LIN {X 0,Y 199.538,Z 723.393,A -85,B 0,C 180,E1 -21434.273,E2 -21434.273} C_VEL
LIN {X 0,Y 200.491,Z 712.919,A -85,B 0,C 180,E1 -21436.81,E2 -21436.81} C_VEL
LIN {X 0,Y 201.96,Z 700.232,A -85,B 0,C 180,E1 -21439.305,E2 -21439.305} C_VEL
LIN {X 0,Y 203.313,Z 687.711,A -85,B 0,C 180,E1 -21441.281,E2 -21441.281} C_VEL
LIN {X 0,Y 204.53,Z 673.735,A -85,B 0,C 180,E1 -21443.008,E2 -21443.008} C_VEL
LIN {X 0,Y 205.706,Z 659.307,A -85,B 0,C 180,E1 -21444.338,E2 -21444.338} C_VEL
LIN {X 0,Y 207.39,Z 632.291,A -85,B 0,C 180,E1 -21446.071,E2 -21446.071} C_VEL
LIN {X 0,Y 210.434,Z 583.695,A -85,B 0,C 180,E1 -21448.978,E2 -21448.978} C_VEL
LIN {X 0,Y 207.804,Z 555.517,A -85,B 0,C 180,E1 -21450.892,E2 -21450.892} C_VEL
LIN {X 0,Y 206.873,Z 542.727,A -85,B 0,C 180,E1 -21451.758,E2 -21451.758} C_VEL
LIN {X 0,Y 205.476,Z 537.587,A -85,B 0,C 180,E1 -21452.224,E2 -21452.224} C_VEL
LIN {X 0,Y 203.171,Z 526.588,A -85,B 0,C 180,E1 -21456.553,E2 -21456.553} C_VEL
LIN {X 0,Y 200.78,Z 515.899,A -85,B 0,C 180,E1 -21461,E2 -21461} C_VEL
LIN {X 0,Y 199.612,Z 510.746,A -85,B 0,C 180,E1 -21463.319,E2 -21463.319} C_VEL
LIN {X 0,Y 199.581,Z 510.751,A -85,B 0,C 180,E1 -21468.005,E2 -21468.005} C_VEL
LIN {X 0,Y 199.612,Z 510.744,A -85,B 0,C 180,E1 -21470.767,E2 -21470.767} C_VEL
LIN {X 0,Y 199.616,Z 510.742,A -85,B 0,C 180,E1 -21475.714,E2 -21475.714} C_VEL
LIN {X 0,Y 199.703,Z 510.733,A -85,B 0,C 180,E1 -21478.137,E2 -21478.137} C_VEL
LIN {X 0,Y 199.688,Z 510.733,A -85,B 0,C 180,E1 -21482.772,E2 -21482.772} C_VEL
LIN {X 0,Y 199.74,Z 510.729,A -85,B 0,C 180,E1 -21487.229,E2 -21487.229} C_VEL
LIN {X 0,Y 199.798,Z 510.719,A -85,B 0,C 180,E1 -21491.757,E2 -21491.757} C_VEL
LIN {X 0,Y 199.85,Z 510.716,A -85,B 0,C 180,E1 -21495.749,E2 -21495.749} C_VEL
LIN {X 0,Y 200.077,Z 510.684,A -85,B 0,C 180,E1 -21499.884,E2 -21499.884} C_VEL
LIN {X 0,Y 200.134,Z 510.678,A -85,B 0,C 180,E1 -21501.925,E2 -21501.925} C_VEL
LIN {X 0,Y 200.326,Z 510.653,A -85,B 0,C 180,E1 -21507.989,E2 -21507.989} C_VEL
LIN {X 0,Y 200.485,Z 510.633,A -85,B 0,C 180,E1 -21510,E2 -21510} C_VEL
LIN {X 0,Y 200.035,Z 510.692,A -85,B 0,C 180,E1 -21514.029,E2 -21514.029} C_VEL
LIN {X 0,Y 200.134,Z 510.675,A -85,B 0,C 180,E1 -21518.075,E2 -21518.075} C_VEL
LIN {X 0,Y 199.916,Z 510.706,A -85,B 0,C 180,E1 -21522.177,E2 -21522.177} C_VEL
LIN {X 0,Y 199.807,Z 510.716,A -85,B 0,C 180,E1 -21526.343,E2 -21526.343} C_VEL
LIN {X 0,Y 199.825,Z 510.716,A -85,B 0,C 180,E1 -21528.454,E2 -21528.454} C_VEL
LIN {X 0,Y 199.738,Z 510.726,A -85,B 0,C 180,E1 -21533.817,E2 -21533.817} C_VEL
LIN {X 0,Y 199.709,Z 510.731,A -85,B 0,C 180,E1 -21538.384,E2 -21538.384} C_VEL
LIN {X 0,Y 199.659,Z 510.736,A -85,B 0,C 180,E1 -21542.349,E2 -21542.349} C_VEL
LIN {X 0,Y 199.641,Z 510.74,A -85,B 0,C 180,E1 -21546.759,E2 -21546.759} C_VEL
LIN {X 0,Y 199.64,Z 510.743,A -85,B 0,C 180,E1 -21549.321,E2 -21549.321} C_VEL
LIN {X 0,Y 199.583,Z 510.747,A -85,B 0,C 180,E1 -21554.771,E2 -21554.771} C_VEL
LIN {X 0,Y 199.704,Z 510.844,A -85,B 0,C 180,E1 -21560.294,E2 -21560.294} C_VEL
LIN {X 0,Y 203.098,Z 525.538,A -85,B 0,C 180,E1 -21564.592,E2 -21564.592} C_VEL
LIN {X 0,Y 206.826,Z 542.586,A -85,B 0,C 180,E1 -21569.356,E2 -21569.356} C_VEL
LIN {X 0,Y 205.704,Z 551.793,A -85,B 0,C 180,E1 -21571.639,E2 -21571.639} C_VEL
LIN {X 0,Y 207.348,Z 576.297,A -85,B 0,C 180,E1 -21573.193,E2 -21573.193} C_VEL
LIN {X 0,Y 208.243,Z 586.426,A -85,B 0,C 180,E1 -21573.836,E2 -21573.836} C_VEL
LIN {X 0,Y 204.55,Z 659.312,A -85,B 0,C 180,E1 -21578.195,E2 -21578.195} C_VEL
LIN {X 0,Y 203.772,Z 672.943,A -85,B 0,C 180,E1 -21579.255,E2 -21579.255} C_VEL
LIN {X 0,Y 202.728,Z 687.033,A -85,B 0,C 180,E1 -21580.771,E2 -21580.771} C_VEL
LIN {X 0,Y 201.448,Z 700.836,A -85,B 0,C 180,E1 -21582.75,E2 -21582.75} C_VEL
LIN {X 0,Y 200.524,Z 711.943,A -85,B 0,C 180,E1 -21584.76,E2 -21584.76} C_VEL
LIN {X 0,Y 199.491,Z 723.222,A -85,B 0,C 180,E1 -21587.28,E2 -21587.28} C_VEL
LIN {X 0,Y 198.722,Z 732.467,A -85,B 0,C 180,E1 -21589.815,E2 -21589.815} C_VEL
LIN {X 0,Y 198.121,Z 741.455,A -85,B 0,C 180,E1 -21592.869,E2 -21592.869} C_VEL
LIN {X 0,Y 197.748,Z 748.732,A -85,B 0,C 180,E1 -21595.924,E2 -21595.924} C_VEL
LIN {X 0,Y 197.616,Z 754.553,A -85,B 0,C 180,E1 -21598.981,E2 -21598.981} C_VEL
LIN {X 0,Y 197.613,Z 759.139,A -85,B 0,C 180,E1 -21602.038,E2 -21602.038} C_VEL
LIN {X 0,Y 197.951,Z 763.564,A -85,B 0,C 180,E1 -21606.114,E2 -21606.114} C_VEL
LIN {X 0,Y 198.53,Z 765.19,A -85,B 0,C 180,E1 -21608.141,E2 -21608.141} C_VEL
LIN {X 0,Y 200.16,Z 767.195,A -85,B 0,C 180,E1 -21612.162,E2 -21612.162} C_VEL
LIN {X 0,Y 202.917,Z 767.735,A -85,B 0,C 180,E1 -21616.086,E2 -21616.086} C_VEL
LIN {X 0,Y 206.512,Z 766.801,A -85,B 0,C 180,E1 -21619.896,E2 -21619.896} C_VEL
LIN {X 0,Y 211.438,Z 764.341,A -85,B 0,C 180,E1 -21623.508,E2 -21623.508} C_VEL
LIN {X 0,Y 215.761,Z 761.475,A -85,B 0,C 180,E1 -21626.087,E2 -21626.087} C_VEL
LIN {X 0,Y 220.617,Z 757.719,A -85,B 0,C 180,E1 -21628.545,E2 -21628.545} C_VEL
LIN {X 0,Y 227.825,Z 751.158,A -85,B 0,C 180,E1 -21631.629,E2 -21631.629} C_VEL
LIN {X 0,Y 233.763,Z 744.904,A -85,B 0,C 180,E1 -21633.793,E2 -21633.793} C_VEL
LIN {X 0,Y 241.273,Z 736.006,A -85,B 0,C 180,E1 -21636.147,E2 -21636.147} C_VEL
LIN {X 0,Y 248.109,Z 726.715,A -85,B 0,C 180,E1 -21638.032,E2 -21638.032} C_VEL
LIN {X 0,Y 254.857,Z 716.208,A -85,B 0,C 180,E1 -21639.646,E2 -21639.646} C_VEL
LIN {X 0,Y 261.182,Z 704.933,A -85,B 0,C 180,E1 -21640.987,E2 -21640.987} C_VEL
LIN {X 0,Y 263.869,Z 699.471,A -85,B 0,C 180,E1 -21641.52,E2 -21641.52} C_VEL
LIN {X 0,Y 264.318,Z 698.406,A -85,B 0,C 180,E1 -21641.773,E2 -21641.773} C_VEL
LIN {X 0,Y 264.338,Z 697.972,A -85,B 0,C 180,E1 -21642.395,E2 -21642.395} C_VEL
LIN {X 0,Y 263.457,Z 699.205,A -85,B 0,C 180,E1 -21643.374,E2 -21643.374} C_VEL
LIN {X 0,Y 262.431,Z 700.943,A -85,B 0,C 180,E1 -21644.031,E2 -21644.031} C_VEL
LIN {X 0,Y 259.901,Z 705.499,A -85,B 0,C 180,E1 -21645.208,E2 -21645.208} C_VEL
LIN {X 0,Y 257.019,Z 710.646,A -85,B 0,C 180,E1 -21646.213,E2 -21646.213} C_VEL
LIN {X 0,Y 254.784,Z 714.396,A -85,B 0,C 180,E1 -21646.735,E2 -21646.735} C_VEL
LIN {X 0,Y 247.204,Z 725.947,A -85,B 0,C 180,E1 -21648.238,E2 -21648.238} C_VEL
LIN {X 0,Y 238.723,Z 737.138,A -85,B 0,C 180,E1 -21650.184,E2 -21650.184} C_VEL
LIN {X 0,Y 231.018,Z 746.108,A -85,B 0,C 180,E1 -21652.276,E2 -21652.276} C_VEL
LIN {X 0,Y 223.904,Z 753.524,A -85,B 0,C 180,E1 -21654.501,E2 -21654.501} C_VEL
LIN {X 0,Y 217.848,Z 759.259,A -85,B 0,C 180,E1 -21656.74,E2 -21656.74} C_VEL
LIN {X 0,Y 210.681,Z 765.375,A -85,B 0,C 180,E1 -21659.975,E2 -21659.975} C_VEL
LIN {X 0,Y 204.411,Z 769.92,A -85,B 0,C 180,E1 -21663.451,E2 -21663.451} C_VEL
LIN {X 0,Y 199.387,Z 773.014,A -85,B 0,C 180,E1 -21667.187,E2 -21667.187} C_VEL
LIN {X 0,Y 195.455,Z 774.755,A -85,B 0,C 180,E1 -21671.118,E2 -21671.118} C_VEL
LIN {X 0,Y 192.647,Z 775.104,A -85,B 0,C 180,E1 -21675.205,E2 -21675.205} C_VEL
LIN {X 0,Y 191.118,Z 774.041,A -85,B 0,C 180,E1 -21679.405,E2 -21679.405} C_VEL
LIN {X 0,Y 190.659,Z 771.533,A -85,B 0,C 180,E1 -21683.651,E2 -21683.651} C_VEL
LIN {X 0,Y 190.784,Z 768.594,A -85,B 0,C 180,E1 -21686.833,E2 -21686.833} C_VEL
LIN {X 0,Y 191.06,Z 766.027,A -85,B 0,C 180,E1 -21689.078,E2 -21689.078} C_VEL
LIN {X 0,Y 190.744,Z 769.407,A -85,B 0,C 180,E1 -21692.112,E2 -21692.112} C_VEL
LIN {X 0,Y 190.574,Z 772.03,A -85,B 0,C 180,E1 -21695.311,E2 -21695.311} C_VEL
LIN {X 0,Y 190.623,Z 773.843,A -85,B 0,C 180,E1 -21698.481,E2 -21698.481} C_VEL
LIN {X 0,Y 191.584,Z 775.164,A -85,B 0,C 180,E1 -21702.715,E2 -21702.715} C_VEL
LIN {X 0,Y 193.65,Z 775.273,A -85,B 0,C 180,E1 -21706.878,E2 -21706.878} C_VEL
LIN {X 0,Y 196.855,Z 774.188,A -85,B 0,C 180,E1 -21710.917,E2 -21710.917} C_VEL
LIN {X 0,Y 201.1,Z 771.909,A -85,B 0,C 180,E1 -21714.795,E2 -21714.795} C_VEL
LIN {X 0,Y 206.36,Z 768.461,A -85,B 0,C 180,E1 -21718.477,E2 -21718.477} C_VEL
LIN {X 0,Y 212.807,Z 763.716,A -85,B 0,C 180,E1 -21721.898,E2 -21721.898} C_VEL
LIN {X 0,Y 220.248,Z 757.558,A -85,B 0,C 180,E1 -21725.056,E2 -21725.056} C_VEL
LIN {X 0,Y 227.423,Z 751.033,A -85,B 0,C 180,E1 -21727.614,E2 -21727.614} C_VEL
LIN {X 0,Y 236.499,Z 741.882,A -85,B 0,C 180,E1 -21730.267,E2 -21730.267} C_VEL
LIN {X 0,Y 243.795,Z 733.654,A -85,B 0,C 180,E1 -21732.086,E2 -21732.086} C_VEL
LIN {X 0,Y 252.794,Z 722.394,A -85,B 0,C 180,E1 -21734.03,E2 -21734.03} C_VEL
LIN {X 0,Y 261.497,Z 709.921,A -85,B 0,C 180,E1 -21735.627,E2 -21735.627} C_VEL
LIN {X 0,Y 267.73,Z 699.805,A -85,B 0,C 180,E1 -21736.599,E2 -21736.599} C_VEL
LIN {X 0,Y 269.637,Z 696.414,A -85,B 0,C 180,E1 -21736.871,E2 -21736.871} C_VEL
LIN {X 0,Y 268.965,Z 697.521,A -85,B 0,C 180,E1 -21737.205,E2 -21737.205} C_VEL
LIN {X 0,Y 261.172,Z 710.023,A -85,B 0,C 180,E1 -21738.498,E2 -21738.498} C_VEL
LIN {X 0,Y 252.468,Z 722.025,A -85,B 0,C 180,E1 -21740.189,E2 -21740.189} C_VEL
LIN {X 0,Y 244.82,Z 731.27,A -85,B 0,C 180,E1 -21741.888,E2 -21741.888} C_VEL
LIN {X 0,Y 236.371,Z 740.349,A -85,B 0,C 180,E1 -21744.04,E2 -21744.04} C_VEL
LIN {X 0,Y 227.276,Z 748.967,A -85,B 0,C 180,E1 -21746.829,E2 -21746.829} C_VEL
LIN {X 0,Y 220.355,Z 754.627,A -85,B 0,C 180,E1 -21749.316,E2 -21749.316} C_VEL
LIN {X 0,Y 214.842,Z 758.693,A -85,B 0,C 180,E1 -21751.684,E2 -21751.684} C_VEL
LIN {X 0,Y 209.813,Z 761.867,A -85,B 0,C 180,E1 -21754.186,E2 -21754.186} C_VEL
LIN {X 0,Y 204.001,Z 764.903,A -85,B 0,C 180,E1 -21757.731,E2 -21757.731} C_VEL
LIN {X 0,Y 199.095,Z 766.562,A -85,B 0,C 180,E1 -21761.476,E2 -21761.476} C_VEL
LIN {X 0,Y 195.476,Z 766.806,A -85,B 0,C 180,E1 -21765.423,E2 -21765.423} C_VEL
LIN {X 0,Y 192.791,Z 765.642,A -85,B 0,C 180,E1 -21769.498,E2 -21769.498} C_VEL
LIN {X 0,Y 191.187,Z 763.064,A -85,B 0,C 180,E1 -21773.669,E2 -21773.669} C_VEL
LIN {X 0,Y 190.614,Z 758.971,A -85,B 0,C 180,E1 -21777.887,E2 -21777.887} C_VEL
LIN {X 0,Y 190.501,Z 754.761,A -85,B 0,C 180,E1 -21781.057,E2 -21781.057} C_VEL
LIN {X 0,Y 190.533,Z 749.385,A -85,B 0,C 180,E1 -21784.231,E2 -21784.231} C_VEL
LIN {X 0,Y 190.87,Z 742.738,A -85,B 0,C 180,E1 -21787.404,E2 -21787.404} C_VEL
LIN {X 0,Y 191.407,Z 734.574,A -85,B 0,C 180,E1 -21790.579,E2 -21790.579} C_VEL
LIN {X 0,Y 192.322,Z 724.548,A -85,B 0,C 180,E1 -21793.741,E2 -21793.741} C_VEL
LIN {X 0,Y 193.237,Z 714.276,A -85,B 0,C 180,E1 -21796.372,E2 -21796.372} C_VEL
LIN {X 0,Y 194.667,Z 701.848,A -85,B 0,C 180,E1 -21798.961,E2 -21798.961} C_VEL
LIN {X 0,Y 196.017,Z 689.687,A -85,B 0,C 180,E1 -21801.011,E2 -21801.011} C_VEL
LIN {X 0,Y 197.215,Z 676.294,A -85,B 0,C 180,E1 -21802.801,E2 -21802.801} C_VEL
LIN {X 0,Y 198.466,Z 661.566,A -85,B 0,C 180,E1 -21804.309,E2 -21804.309} C_VEL
LIN {X 0,Y 199.852,Z 640.548,A -85,B 0,C 180,E1 -21805.797,E2 -21805.797} C_VEL
LIN {X 0,Y 203.424,Z 584.022,A -85,B 0,C 180,E1 -21809.337,E2 -21809.337} C_VEL
LIN {X 0,Y 200.675,Z 552.776,A -85,B 0,C 180,E1 -21811.545,E2 -21811.545} C_VEL
LIN {X 0,Y 200.037,Z 544.275,A -85,B 0,C 180,E1 -21812.141,E2 -21812.141} C_VEL
LIN {X 0,Y 198.245,Z 537.538,A -85,B 0,C 180,E1 -21812.733,E2 -21812.733} C_VEL
LIN {X 0,Y 195.977,Z 526.924,A -85,B 0,C 180,E1 -21817.07,E2 -21817.07} C_VEL
LIN {X 0,Y 193.455,Z 515.636,A -85,B 0,C 180,E1 -21821.947,E2 -21821.947} C_VEL
LIN {X 0,Y 192.558,Z 511.625,A -85,B 0,C 180,E1 -21823.748,E2 -21823.748} C_VEL
LIN {X 0,Y 192.515,Z 511.63,A -85,B 0,C 180,E1 -21828.92,E2 -21828.92} C_VEL
LIN {X 0,Y 192.588,Z 511.621,A -85,B 0,C 180,E1 -21833.402,E2 -21833.402} C_VEL
LIN {X 0,Y 192.612,Z 511.614,A -85,B 0,C 180,E1 -21837.058,E2 -21837.058} C_VEL
LIN {X 0,Y 192.666,Z 511.61,A -85,B 0,C 180,E1 -21841.692,E2 -21841.692} C_VEL
LIN {X 0,Y 192.707,Z 511.603,A -85,B 0,C 180,E1 -21846.349,E2 -21846.349} C_VEL
LIN {X 0,Y 192.733,Z 511.6,A -85,B 0,C 180,E1 -21851.457,E2 -21851.457} C_VEL
LIN {X 0,Y 192.774,Z 511.596,A -85,B 0,C 180,E1 -21855.214,E2 -21855.214} C_VEL
LIN {X 0,Y 193.022,Z 511.565,A -85,B 0,C 180,E1 -21859.51,E2 -21859.51} C_VEL
LIN {X 0,Y 193.007,Z 511.568,A -85,B 0,C 180,E1 -21863.728,E2 -21863.728} C_VEL
LIN {X 0,Y 193.268,Z 511.533,A -85,B 0,C 180,E1 -21867.916,E2 -21867.916} C_VEL
LIN {X 0,Y 193.448,Z 511.509,A -85,B 0,C 180,E1 -21870,E2 -21870} C_VEL
LIN {X 0,Y 192.982,Z 511.57,A -85,B 0,C 180,E1 -21874.177,E2 -21874.177} C_VEL
LIN {X 0,Y 193.081,Z 511.553,A -85,B 0,C 180,E1 -21878.372,E2 -21878.372} C_VEL
LIN {X 0,Y 192.855,Z 511.586,A -85,B 0,C 180,E1 -21882.63,E2 -21882.63} C_VEL
LIN {X 0,Y 192.782,Z 511.593,A -85,B 0,C 180,E1 -21888.586,E2 -21888.586} C_VEL
LIN {X 0,Y 192.665,Z 511.606,A -85,B 0,C 180,E1 -21894.225,E2 -21894.225} C_VEL
LIN {X 0,Y 192.645,Z 511.612,A -85,B 0,C 180,E1 -21898.889,E2 -21898.889} C_VEL
LIN {X 0,Y 192.599,Z 511.616,A -85,B 0,C 180,E1 -21903.186,E2 -21903.186} C_VEL
LIN {X 0,Y 192.61,Z 511.616,A -85,B 0,C 180,E1 -21906.608,E2 -21906.608} C_VEL
LIN {X 0,Y 192.525,Z 511.627,A -85,B 0,C 180,E1 -21911.077,E2 -21911.077} C_VEL
LIN {X 0,Y 192.494,Z 511.631,A -85,B 0,C 180,E1 -21916.077,E2 -21916.077} C_VEL
LIN {X 0,Y 192.647,Z 511.756,A -85,B 0,C 180,E1 -21919.857,E2 -21919.857} C_VEL
LIN {X 0,Y 196.065,Z 526.547,A -85,B 0,C 180,E1 -21924.291,E2 -21924.291} C_VEL
LIN {X 0,Y 199.703,Z 543.053,A -85,B 0,C 180,E1 -21929.027,E2 -21929.027} C_VEL
LIN {X 0,Y 198.736,Z 551.747,A -85,B 0,C 180,E1 -21931.279,E2 -21931.279} C_VEL
LIN {X 0,Y 200.206,Z 575.588,A -85,B 0,C 180,E1 -21932.848,E2 -21932.848} C_VEL
LIN {X 0,Y 201.175,Z 587.238,A -85,B 0,C 180,E1 -21933.62,E2 -21933.62} C_VEL
LIN {X 0,Y 197.436,Z 659.441,A -85,B 0,C 180,E1 -21938.166,E2 -21938.166} C_VEL
LIN {X 0,Y 196.622,Z 673.729,A -85,B 0,C 180,E1 -21939.331,E2 -21939.331} C_VEL
LIN {X 0,Y 195.6,Z 687.334,A -85,B 0,C 180,E1 -21940.861,E2 -21940.861} C_VEL
LIN {X 0,Y 194.328,Z 701.111,A -85,B 0,C 180,E1 -21942.912,E2 -21942.912} C_VEL
LIN {X 0,Y 193.391,Z 712.142,A -85,B 0,C 180,E1 -21944.994,E2 -21944.994} C_VEL
LIN {X 0,Y 192.369,Z 723.29,A -85,B 0,C 180,E1 -21947.606,E2 -21947.606} C_VEL
LIN {X 0,Y 191.583,Z 733.292,A -85,B 0,C 180,E1 -21950.498,E2 -21950.498} C_VEL
LIN {X 0,Y 191.032,Z 742.187,A -85,B 0,C 180,E1 -21953.663,E2 -21953.663} C_VEL
LIN {X 0,Y 190.726,Z 749.346,A -85,B 0,C 180,E1 -21956.832,E2 -21956.832} C_VEL
LIN {X 0,Y 190.588,Z 755.01,A -85,B 0,C 180,E1 -21960,E2 -21960} C_VEL
LIN {X 0,Y 190.61,Z 759.489,A -85,B 0,C 180,E1 -21963.171,E2 -21963.171} C_VEL
LIN {X 0,Y 190.924,Z 762.954,A -85,B 0,C 180,E1 -21966.34,E2 -21966.34} C_VEL
LIN {X 0,Y 192.242,Z 766.101,A -85,B 0,C 180,E1 -21970.532,E2 -21970.532} C_VEL
LIN {X 0,Y 194.54,Z 767.777,A -85,B 0,C 180,E1 -21974.648,E2 -21974.648} C_VEL
LIN {X 0,Y 197.887,Z 767.941,A -85,B 0,C 180,E1 -21978.641,E2 -21978.641} C_VEL
LIN {X 0,Y 199.901,Z 767.499,A -85,B 0,C 180,E1 -21980.584,E2 -21980.584} C_VEL
LIN {X 0,Y 205.058,Z 765.507,A -85,B 0,C 180,E1 -21984.285,E2 -21984.285} C_VEL
LIN {X 0,Y 207.958,Z 763.962,A -85,B 0,C 180,E1 -21986.062,E2 -21986.062} C_VEL
LIN {X 0,Y 214.603,Z 759.634,A -85,B 0,C 180,E1 -21989.422,E2 -21989.422} C_VEL
LIN {X 0,Y 220.177,Z 755.324,A -85,B 0,C 180,E1 -21991.781,E2 -21991.781} C_VEL
LIN {X 0,Y 227.232,Z 749.022,A -85,B 0,C 180,E1 -21994.364,E2 -21994.364} C_VEL
LIN {X 0,Y 234.899,Z 741.08,A -85,B 0,C 180,E1 -21996.754,E2 -21996.754} C_VEL
LIN {X 0,Y 241.856,Z 732.883,A -85,B 0,C 180,E1 -21998.665,E2 -21998.665} C_VEL
LIN {X 0,Y 249.347,Z 722.876,A -85,B 0,C 180,E1 -22000.411,E2 -22000.411} C_VEL
LIN {X 0,Y 256.515,Z 711.735,A -85,B 0,C 180,E1 -22001.9,E2 -22001.9} C_VEL
LIN {X 0,Y 262.946,Z 700.024,A -85,B 0,C 180,E1 -22003.08,E2 -22003.08} C_VEL
LIN {X 0,Y 268.228,Z 688.618,A -85,B 0,C 180,E1 -22003.975,E2 -22003.975} C_VEL
LIN {X 0,Y 269.024,Z 686.717,A -85,B 0,C 180,E1 -22004.102,E2 -22004.102} C_VEL
LIN {X 0,Y 269.42,Z 685.699,A -85,B 0,C 180,E1 -22004.443,E2 -22004.443} C_VEL
LIN {X 0,Y 263.476,Z 698.717,A -85,B 0,C 180,E1 -22005.289,E2 -22005.289} C_VEL
LIN {X 0,Y 257.055,Z 710.637,A -85,B 0,C 180,E1 -22006.342,E2 -22006.342} C_VEL
LIN {X 0,Y 254.784,Z 714.396,A -85,B 0,C 180,E1 -22006.735,E2 -22006.735} C_VEL
LIN {X 0,Y 251.69,Z 719.15,A -85,B 0,C 180,E1 -22007.147,E2 -22007.147} C_VEL
LIN {X 0,Y 245.838,Z 727.009,A -85,B 0,C 180,E1 -22007.524,E2 -22007.524} C_VEL
LIN {X 0,Y 239.679,Z 734.365,A -85,B 0,C 180,E1 -22008.005,E2 -22008.005} C_VEL
LIN {X 0,Y 236.142,Z 738.329,A -85,B 0,C 180,E1 -22008.587,E2 -22008.587} C_VEL
LIN {X 0,Y 227.616,Z 747.405,A -85,B 0,C 180,E1 -22010.73,E2 -22010.73} C_VEL
LIN {X 0,Y 220.62,Z 754.006,A -85,B 0,C 180,E1 -22012.752,E2 -22012.752} C_VEL
LIN {X 0,Y 214.164,Z 759.568,A -85,B 0,C 180,E1 -22014.951,E2 -22014.951} C_VEL
LIN {X 0,Y 208.291,Z 764.134,A -85,B 0,C 180,E1 -22017.326,E2 -22017.326} C_VEL
LIN {X 0,Y 201.283,Z 768.901,A -85,B 0,C 180,E1 -22020.737,E2 -22020.737} C_VEL
LIN {X 0,Y 195.34,Z 772.234,A -85,B 0,C 180,E1 -22024.422,E2 -22024.422} C_VEL
LIN {X 0,Y 190.648,Z 774.189,A -85,B 0,C 180,E1 -22028.368,E2 -22028.368} C_VEL
LIN {X 0,Y 187.113,Z 774.819,A -85,B 0,C 180,E1 -22032.514,E2 -22032.514} C_VEL
LIN {X 0,Y 184.858,Z 774.114,A -85,B 0,C 180,E1 -22036.814,E2 -22036.814} C_VEL
LIN {X 0,Y 183.783,Z 771.993,A -85,B 0,C 180,E1 -22041.201,E2 -22041.201} C_VEL
LIN {X 0,Y 183.786,Z 768.349,A -85,B 0,C 180,E1 -22045.614,E2 -22045.614} C_VEL
LIN {X 0,Y 184.114,Z 764.515,A -85,B 0,C 180,E1 -22049.043,E2 -22049.043} C_VEL
LIN {X 0,Y 183.694,Z 769.129,A -85,B 0,C 180,E1 -22053.29,E2 -22053.29} C_VEL
LIN {X 0,Y 183.514,Z 771.696,A -85,B 0,C 180,E1 -22056.597,E2 -22056.597} C_VEL
LIN {X 0,Y 184.062,Z 773.925,A -85,B 0,C 180,E1 -22061.006,E2 -22061.006} C_VEL
LIN {X 0,Y 185.559,Z 774.936,A -85,B 0,C 180,E1 -22065.375,E2 -22065.375} C_VEL
LIN {X 0,Y 188.401,Z 774.77,A -85,B 0,C 180,E1 -22069.617,E2 -22069.617} C_VEL
LIN {X 0,Y 192.278,Z 773.441,A -85,B 0,C 180,E1 -22073.708,E2 -22073.708} C_VEL
LIN {X 0,Y 197.392,Z 770.954,A -85,B 0,C 180,E1 -22077.572,E2 -22077.572} C_VEL
LIN {X 0,Y 203.443,Z 767.313,A -85,B 0,C 180,E1 -22081.21,E2 -22081.21} C_VEL
LIN {X 0,Y 210.669,Z 762.373,A -85,B 0,C 180,E1 -22084.55,E2 -22084.55} C_VEL
LIN {X 0,Y 218.805,Z 756.107,A -85,B 0,C 180,E1 -22087.61,E2 -22087.61} C_VEL
LIN {X 0,Y 227.831,Z 748.331,A -85,B 0,C 180,E1 -22090.376,E2 -22090.376} C_VEL
LIN {X 0,Y 237.647,Z 738.718,A -85,B 0,C 180,E1 -22092.859,E2 -22092.859} C_VEL
LIN {X 0,Y 245.49,Z 730.127,A -85,B 0,C 180,E1 -22094.54,E2 -22094.54} C_VEL
LIN {X 0,Y 253.719,Z 720.134,A -85,B 0,C 180,E1 -22096.071,E2 -22096.071} C_VEL
LIN {X 0,Y 259.381,Z 712.449,A -85,B 0,C 180,E1 -22097.019,E2 -22097.019} C_VEL
LIN {X 0,Y 254.554,Z 718.823,A -85,B 0,C 180,E1 -22097.917,E2 -22097.917} C_VEL
LIN {X 0,Y 246.269,Z 728.621,A -85,B 0,C 180,E1 -22099.516,E2 -22099.516} C_VEL
LIN {X 0,Y 237.221,Z 738.14,A -85,B 0,C 180,E1 -22101.526,E2 -22101.526} C_VEL
LIN {X 0,Y 228.736,Z 745.987,A -85,B 0,C 180,E1 -22103.739,E2 -22103.739} C_VEL
LIN {X 0,Y 220.253,Z 752.791,A -85,B 0,C 180,E1 -22106.333,E2 -22106.333} C_VEL
LIN {X 0,Y 212.546,Z 758.198,A -85,B 0,C 180,E1 -22109.168,E2 -22109.168} C_VEL
LIN {X 0,Y 206.989,Z 761.576,A -85,B 0,C 180,E1 -22111.618,E2 -22111.618} C_VEL
LIN {X 0,Y 200.447,Z 764.78,A -85,B 0,C 180,E1 -22115.119,E2 -22115.119} C_VEL
LIN {X 0,Y 194.867,Z 766.667,A -85,B 0,C 180,E1 -22118.859,E2 -22118.859} C_VEL
LIN {X 0,Y 190.322,Z 767.202,A -85,B 0,C 180,E1 -22122.817,E2 -22122.817} C_VEL
LIN {X 0,Y 187.097,Z 766.38,A -85,B 0,C 180,E1 -22126.975,E2 -22126.975} C_VEL
LIN {X 0,Y 184.841,Z 764.169,A -85,B 0,C 180,E1 -22131.252,E2 -22131.252} C_VEL
LIN {X 0,Y 183.796,Z 760.491,A -85,B 0,C 180,E1 -22135.614,E2 -22135.614} C_VEL
LIN {X 0,Y 183.525,Z 756.679,A -85,B 0,C 180,E1 -22138.903,E2 -22138.903} C_VEL
LIN {X 0,Y 183.469,Z 751.805,A -85,B 0,C 180,E1 -22142.195,E2 -22142.195} C_VEL
LIN {X 0,Y 183.677,Z 745.06,A -85,B 0,C 180,E1 -22145.822,E2 -22145.822} C_VEL
LIN {X 0,Y 184.183,Z 736.79,A -85,B 0,C 180,E1 -22149.333,E2 -22149.333} C_VEL
LIN {X 0,Y 184.937,Z 727.264,A -85,B 0,C 180,E1 -22152.622,E2 -22152.622} C_VEL
LIN {X 0,Y 185.945,Z 716.545,A -85,B 0,C 180,E1 -22155.622,E2 -22155.622} C_VEL
LIN {X 0,Y 187.18,Z 704.739,A -85,B 0,C 180,E1 -22158.328,E2 -22158.328} C_VEL
LIN {X 0,Y 188.61,Z 692.172,A -85,B 0,C 180,E1 -22160.624,E2 -22160.624} C_VEL
LIN {X 0,Y 189.911,Z 678.748,A -85,B 0,C 180,E1 -22162.576,E2 -22162.576} C_VEL
LIN {X 0,Y 191.114,Z 664.628,A -85,B 0,C 180,E1 -22164.149,E2 -22164.149} C_VEL
LIN {X 0,Y 192.222,Z 649.678,A -85,B 0,C 180,E1 -22165.37,E2 -22165.37} C_VEL
LIN {X 0,Y 196.444,Z 584.623,A -85,B 0,C 180,E1 -22169.68,E2 -22169.68} C_VEL
LIN {X 0,Y 193.939,Z 555.999,A -85,B 0,C 180,E1 -22171.772,E2 -22171.772} C_VEL
LIN {X 0,Y 193.238,Z 546.026,A -85,B 0,C 180,E1 -22172.5,E2 -22172.5} C_VEL
LIN {X 0,Y 190.956,Z 537.385,A -85,B 0,C 180,E1 -22173.306,E2 -22173.306} C_VEL
LIN {X 0,Y 188.38,Z 525.374,A -85,B 0,C 180,E1 -22178.421,E2 -22178.421} C_VEL
LIN {X 0,Y 186.035,Z 514.853,A -85,B 0,C 180,E1 -22183.167,E2 -22183.167} C_VEL
LIN {X 0,Y 185.496,Z 512.504,A -85,B 0,C 180,E1 -22184.357,E2 -22184.357} C_VEL
LIN {X 0,Y 185.47,Z 512.508,A -85,B 0,C 180,E1 -22189.895,E2 -22189.895} C_VEL
LIN {X 0,Y 185.507,Z 512.501,A -85,B 0,C 180,E1 -22192.711,E2 -22192.711} C_VEL
LIN {X 0,Y 185.548,Z 512.496,A -85,B 0,C 180,E1 -22197.975,E2 -22197.975} C_VEL
LIN {X 0,Y 185.583,Z 512.491,A -85,B 0,C 180,E1 -22200.576,E2 -22200.576} C_VEL
LIN {X 0,Y 185.589,Z 512.489,A -85,B 0,C 180,E1 -22205.382,E2 -22205.382} C_VEL
LIN {X 0,Y 185.676,Z 512.48,A -85,B 0,C 180,E1 -22211.133,E2 -22211.133} C_VEL
LIN {X 0,Y 185.726,Z 512.472,A -85,B 0,C 180,E1 -22214.64,E2 -22214.64} C_VEL
LIN {X 0,Y 185.944,Z 512.448,A -85,B 0,C 180,E1 -22219.328,E2 -22219.328} C_VEL
LIN {X 0,Y 185.971,Z 512.444,A -85,B 0,C 180,E1 -22223.49,E2 -22223.49} C_VEL
LIN {X 0,Y 186.212,Z 512.412,A -85,B 0,C 180,E1 -22227.837,E2 -22227.837} C_VEL
LIN {X 0,Y 186.411,Z 512.385,A -85,B 0,C 180,E1 -22230,E2 -22230} C_VEL
LIN {X 0,Y 185.93,Z 512.448,A -85,B 0,C 180,E1 -22234.335,E2 -22234.335} C_VEL
LIN {X 0,Y 186.031,Z 512.431,A -85,B 0,C 180,E1 -22238.691,E2 -22238.691} C_VEL
LIN {X 0,Y 185.767,Z 512.47,A -85,B 0,C 180,E1 -22243.12,E2 -22243.12} C_VEL
LIN {X 0,Y 185.718,Z 512.474,A -85,B 0,C 180,E1 -22247.622,E2 -22247.622} C_VEL
LIN {X 0,Y 185.601,Z 512.489,A -85,B 0,C 180,E1 -22252.251,E2 -22252.251} C_VEL
LIN {X 0,Y 185.561,Z 512.493,A -85,B 0,C 180,E1 -22257.032,E2 -22257.032} C_VEL
LIN {X 0,Y 185.578,Z 512.494,A -85,B 0,C 180,E1 -22259.493,E2 -22259.493} C_VEL
LIN {X 0,Y 185.519,Z 512.496,A -85,B 0,C 180,E1 -22264.628,E2 -22264.628} C_VEL
LIN {X 0,Y 185.545,Z 512.499,A -85,B 0,C 180,E1 -22267.304,E2 -22267.304} C_VEL
LIN {X 0,Y 185.487,Z 512.503,A -85,B 0,C 180,E1 -22270.73,E2 -22270.73} C_VEL
LIN {X 0,Y 185.483,Z 512.503,A -85,B 0,C 180,E1 -22273.953,E2 -22273.953} C_VEL
LIN {X 0,Y 185.567,Z 512.52,A -85,B 0,C 180,E1 -22279.369,E2 -22279.369} C_VEL
LIN {X 0,Y 189.206,Z 528.348,A -85,B 0,C 180,E1 -22284.24,E2 -22284.24} C_VEL
LIN {X 0,Y 192.59,Z 543.697,A -85,B 0,C 180,E1 -22288.747,E2 -22288.747} C_VEL
LIN {X 0,Y 192.152,Z 549.113,A -85,B 0,C 180,E1 -22290.201,E2 -22290.201} C_VEL
LIN {X 0,Y 191.735,Z 551.898,A -85,B 0,C 180,E1 -22290.936,E2 -22290.936} C_VEL
LIN {X 0,Y 193.19,Z 576.268,A -85,B 0,C 180,E1 -22292.624,E2 -22292.624} C_VEL
LIN {X 0,Y 194.111,Z 587.271,A -85,B 0,C 180,E1 -22293.381,E2 -22293.381} C_VEL
LIN {X 0,Y 190.376,Z 658.875,A -85,B 0,C 180,E1 -22298.087,E2 -22298.087} C_VEL
LIN {X 0,Y 189.591,Z 672.752,A -85,B 0,C 180,E1 -22299.239,E2 -22299.239} C_VEL
LIN {X 0,Y 188.479,Z 687.413,A -85,B 0,C 180,E1 -22300.957,E2 -22300.957} C_VEL
LIN {X 0,Y 187.235,Z 701.052,A -85,B 0,C 180,E1 -22303.088,E2 -22303.088} C_VEL
LIN {X 0,Y 186.325,Z 712.08,A -85,B 0,C 180,E1 -22305.25,E2 -22305.25} C_VEL
LIN {X 0,Y 185.276,Z 723.249,A -85,B 0,C 180,E1 -22307.958,E2 -22307.958} C_VEL
LIN {X 0,Y 184.562,Z 732.49,A -85,B 0,C 180,E1 -22310.687,E2 -22310.687} C_VEL
LIN {X 0,Y 184.029,Z 741.513,A -85,B 0,C 180,E1 -22313.977,E2 -22313.977} C_VEL
LIN {X 0,Y 183.731,Z 748.746,A -85,B 0,C 180,E1 -22317.259,E2 -22317.259} C_VEL
LIN {X 0,Y 183.604,Z 753.663,A -85,B 0,C 180,E1 -22320,E2 -22320} C_VEL
LIN {X 0,Y 183.613,Z 758.478,A -85,B 0,C 180,E1 -22323.291,E2 -22323.291} C_VEL
LIN {X 0,Y 183.92,Z 762.172,A -85,B 0,C 180,E1 -22326.583,E2 -22326.583} C_VEL
LIN {X 0,Y 185.292,Z 765.747,A -85,B 0,C 180,E1 -22330.932,E2 -22330.932} C_VEL
LIN {X 0,Y 187.676,Z 767.747,A -85,B 0,C 180,E1 -22335.197,E2 -22335.197} C_VEL
LIN {X 0,Y 191.184,Z 768.346,A -85,B 0,C 180,E1 -22339.32,E2 -22339.32} C_VEL
LIN {X 0,Y 193.322,Z 768.125,A -85,B 0,C 180,E1 -22341.318,E2 -22341.318} C_VEL
LIN {X 0,Y 198.696,Z 766.568,A -85,B 0,C 180,E1 -22345.116,E2 -22345.116} C_VEL
LIN {X 0,Y 205.081,Z 763.546,A -85,B 0,C 180,E1 -22348.671,E2 -22348.671} C_VEL
LIN {X 0,Y 210.53,Z 760.275,A -85,B 0,C 180,E1 -22351.16,E2 -22351.16} C_VEL
LIN {X 0,Y 218.506,Z 754.528,A -85,B 0,C 180,E1 -22354.254,E2 -22354.254} C_VEL
LIN {X 0,Y 227.362,Z 746.874,A -85,B 0,C 180,E1 -22357.068,E2 -22357.068} C_VEL
LIN {X 0,Y 235.64,Z 738.504,A -85,B 0,C 180,E1 -22359.33,E2 -22359.33} C_VEL
LIN {X 0,Y 242.851,Z 730.146,A -85,B 0,C 180,E1 -22361.025,E2 -22361.025} C_VEL
LIN {X 0,Y 250.809,Z 719.667,A -85,B 0,C 180,E1 -22362.632,E2 -22362.632} C_VEL
LIN {X 0,Y 258.517,Z 707.672,A -85,B 0,C 180,E1 -22364.023,E2 -22364.023} C_VEL
LIN {X 0,Y 258.314,Z 708,A -85,B 0,C 180,E1 -22364.423,E2 -22364.423} C_VEL
LIN {X 0,Y 250.363,Z 720.249,A -85,B 0,C 180,E1 -22365.711,E2 -22365.711} C_VEL
LIN {X 0,Y 244.16,Z 728.642,A -85,B 0,C 180,E1 -22366.872,E2 -22366.872} C_VEL
LIN {X 0,Y 236.142,Z 738.329,A -85,B 0,C 180,E1 -22368.587,E2 -22368.587} C_VEL
LIN {X 0,Y 232.44,Z 742.224,A -85,B 0,C 180,E1 -22369.236,E2 -22369.236} C_VEL
LIN {X 0,Y 225.43,Z 748.557,A -85,B 0,C 180,E1 -22370.041,E2 -22370.041} C_VEL
LIN {X 0,Y 218.338,Z 754.194,A -85,B 0,C 180,E1 -22370.994,E2 -22370.994} C_VEL
LIN {X 0,Y 214.569,Z 757.075,A -85,B 0,C 180,E1 -22371.875,E2 -22371.875} C_VEL
LIN {X 0,Y 206.485,Z 763.013,A -85,B 0,C 180,E1 -22374.646,E2 -22374.646} C_VEL
LIN {X 0,Y 198.726,Z 767.907,A -85,B 0,C 180,E1 -22377.962,E2 -22377.962} C_VEL
LIN {X 0,Y 191.905,Z 771.434,A -85,B 0,C 180,E1 -22381.57,E2 -22381.57} C_VEL
LIN {X 0,Y 186.401,Z 773.631,A -85,B 0,C 180,E1 -22385.497,E2 -22385.497} C_VEL
LIN {X 0,Y 182.041,Z 774.495,A -85,B 0,C 180,E1 -22389.668,E2 -22389.668} C_VEL
LIN {X 0,Y 178.932,Z 774.039,A -85,B 0,C 180,E1 -22394.041,E2 -22394.041} C_VEL
LIN {X 0,Y 177.255,Z 772.282,A -85,B 0,C 180,E1 -22398.566,E2 -22398.566} C_VEL
LIN {X 0,Y 176.732,Z 769.099,A -85,B 0,C 180,E1 -22403.148,E2 -22403.148} C_VEL
LIN {X 0,Y 176.967,Z 765.641,A -85,B 0,C 180,E1 -22406.585,E2 -22406.585} C_VEL
LIN {X 0,Y 177.251,Z 762.734,A -85,B 0,C 180,E1 -22408.935,E2 -22408.935} C_VEL
LIN {X 0,Y 176.73,Z 767.791,A -85,B 0,C 180,E1 -22413.42,E2 -22413.42} C_VEL
LIN {X 0,Y 176.53,Z 770.55,A -85,B 0,C 180,E1 -22416.86,E2 -22416.86} C_VEL
LIN {X 0,Y 177.112,Z 773.098,A -85,B 0,C 180,E1 -22421.444,E2 -22421.444} C_VEL
LIN {X 0,Y 178.706,Z 774.409,A -85,B 0,C 180,E1 -22425.98,E2 -22425.98} C_VEL
LIN {X 0,Y 181.698,Z 774.591,A -85,B 0,C 180,E1 -22430.372,E2 -22430.372} C_VEL
LIN {X 0,Y 185.789,Z 773.628,A -85,B 0,C 180,E1 -22434.589,E2 -22434.589} C_VEL
LIN {X 0,Y 191.135,Z 771.533,A -85,B 0,C 180,E1 -22438.556,E2 -22438.556} C_VEL
LIN {X 0,Y 197.466,Z 768.296,A -85,B 0,C 180,E1 -22442.267,E2 -22442.267} C_VEL
LIN {X 0,Y 204.986,Z 763.872,A -85,B 0,C 180,E1 -22445.652,E2 -22445.652} C_VEL
LIN {X 0,Y 213.425,Z 758.142,A -85,B 0,C 180,E1 -22448.731,E2 -22448.731} C_VEL
LIN {X 0,Y 220.319,Z 752.883,A -85,B 0,C 180,E1 -22450.839,E2 -22450.839} C_VEL
LIN {X 0,Y 230.233,Z 744.559,A -85,B 0,C 180,E1 -22453.38,E2 -22453.38} C_VEL
LIN {X 0,Y 240.878,Z 734.28,A -85,B 0,C 180,E1 -22455.631,E2 -22455.631} C_VEL
LIN {X 0,Y 247.979,Z 726.604,A -85,B 0,C 180,E1 -22456.929,E2 -22456.929} C_VEL
LIN {X 0,Y 248.342,Z 726.127,A -85,B 0,C 180,E1 -22457.219,E2 -22457.219} C_VEL
LIN {X 0,Y 238.714,Z 736.043,A -85,B 0,C 180,E1 -22459.075,E2 -22459.075} C_VEL
LIN {X 0,Y 228.293,Z 745.277,A -85,B 0,C 180,E1 -22461.435,E2 -22461.435} C_VEL
LIN {X 0,Y 219.824,Z 751.806,A -85,B 0,C 180,E1 -22463.739,E2 -22463.739} C_VEL
LIN {X 0,Y 213.012,Z 756.426,A -85,B 0,C 180,E1 -22465.883,E2 -22465.883} C_VEL
LIN {X 0,Y 204.716,Z 761.282,A -85,B 0,C 180,E1 -22469.005,E2 -22469.005} C_VEL
LIN {X 0,Y 197.368,Z 764.719,A -85,B 0,C 180,E1 -22472.425,E2 -22472.425} C_VEL
LIN {X 0,Y 191.081,Z 766.803,A -85,B 0,C 180,E1 -22476.135,E2 -22476.135} C_VEL
LIN {X 0,Y 185.721,Z 767.579,A -85,B 0,C 180,E1 -22480.088,E2 -22480.088} C_VEL
LIN {X 0,Y 181.783,Z 767.016,A -85,B 0,C 180,E1 -22484.298,E2 -22484.298} C_VEL
LIN {X 0,Y 178.875,Z 765.11,A -85,B 0,C 180,E1 -22488.67,E2 -22488.67} C_VEL
LIN {X 0,Y 177.138,Z 761.812,A -85,B 0,C 180,E1 -22493.164,E2 -22493.164} C_VEL
LIN {X 0,Y 176.635,Z 758.347,A -85,B 0,C 180,E1 -22496.578,E2 -22496.578} C_VEL
LIN {X 0,Y 176.486,Z 753.941,A -85,B 0,C 180,E1 -22500,E2 -22500} C_VEL
LIN {X 0,Y 176.558,Z 747.287,A -85,B 0,C 180,E1 -22503.994,E2 -22503.994} C_VEL
LIN {X 0,Y 176.902,Z 740.182,A -85,B 0,C 180,E1 -22507.418,E2 -22507.418} C_VEL
LIN {X 0,Y 177.472,Z 731.48,A -85,B 0,C 180,E1 -22510.842,E2 -22510.842} C_VEL
LIN {X 0,Y 178.443,Z 720.639,A -85,B 0,C 180,E1 -22514.25,E2 -22514.25} C_VEL
LIN {X 0,Y 179.458,Z 709.624,A -85,B 0,C 180,E1 -22517.081,E2 -22517.081} C_VEL
LIN {X 0,Y 180.863,Z 697.681,A -85,B 0,C 180,E1 -22519.582,E2 -22519.582} C_VEL
LIN {X 0,Y 182.317,Z 684.238,A -85,B 0,C 180,E1 -22521.848,E2 -22521.848} C_VEL
LIN {X 0,Y 183.604,Z 669.646,A -85,B 0,C 180,E1 -22523.743,E2 -22523.743} C_VEL
LIN {X 0,Y 184.713,Z 655.409,A -85,B 0,C 180,E1 -22525.117,E2 -22525.117} C_VEL
LIN {X 0,Y 189.407,Z 584.81,A -85,B 0,C 180,E1 -22530.03,E2 -22530.03} C_VEL
LIN {X 0,Y 186.82,Z 554.078,A -85,B 0,C 180,E1 -22532.376,E2 -22532.376} C_VEL
LIN {X 0,Y 186.207,Z 546.799,A -85,B 0,C 180,E1 -22532.94,E2 -22532.94} C_VEL
LIN {X 0,Y 183.695,Z 537.263,A -85,B 0,C 180,E1 -22533.873,E2 -22533.873} C_VEL
LIN {X 0,Y 181.556,Z 527.283,A -85,B 0,C 180,E1 -22538.269,E2 -22538.269} C_VEL
LIN {X 0,Y 179.075,Z 516.204,A -85,B 0,C 180,E1 -22543.443,E2 -22543.443} C_VEL
LIN {X 0,Y 178.425,Z 513.385,A -85,B 0,C 180,E1 -22544.846,E2 -22544.846} C_VEL
LIN {X 0,Y 178.405,Z 513.388,A -85,B 0,C 180,E1 -22548.459,E2 -22548.459} C_VEL
LIN {X 0,Y 178.424,Z 513.382,A -85,B 0,C 180,E1 -22553.783,E2 -22553.783} C_VEL
LIN {X 0,Y 178.489,Z 513.372,A -85,B 0,C 180,E1 -22556.547,E2 -22556.547} C_VEL
LIN {X 0,Y 178.524,Z 513.372,A -85,B 0,C 180,E1 -22560.006,E2 -22560.006} C_VEL
LIN {X 0,Y 178.536,Z 513.365,A -85,B 0,C 180,E1 -22564.875,E2 -22564.875} C_VEL
LIN {X 0,Y 178.625,Z 513.357,A -85,B 0,C 180,E1 -22570.783,E2 -22570.783} C_VEL
LIN {X 0,Y 178.667,Z 513.352,A -85,B 0,C 180,E1 -22574.017,E2 -22574.017} C_VEL
LIN {X 0,Y 178.896,Z 513.325,A -85,B 0,C 180,E1 -22579.153,E2 -22579.153} C_VEL
LIN {X 0,Y 178.936,Z 513.319,A -85,B 0,C 180,E1 -22583.233,E2 -22583.233} C_VEL
LIN {X 0,Y 179.158,Z 513.291,A -85,B 0,C 180,E1 -22587.752,E2 -22587.752} C_VEL
LIN {X 0,Y 179.374,Z 513.262,A -85,B 0,C 180,E1 -22590,E2 -22590} C_VEL
LIN {X 0,Y 178.879,Z 513.327,A -85,B 0,C 180,E1 -22594.507,E2 -22594.507} C_VEL
LIN {X 0,Y 178.98,Z 513.311,A -85,B 0,C 180,E1 -22599.037,E2 -22599.037} C_VEL
LIN {X 0,Y 178.69,Z 513.351,A -85,B 0,C 180,E1 -22603.65,E2 -22603.65} C_VEL
LIN {X 0,Y 178.672,Z 513.35,A -85,B 0,C 180,E1 -22608.341,E2 -22608.341} C_VEL
LIN {X 0,Y 178.515,Z 513.373,A -85,B 0,C 180,E1 -22613.184,E2 -22613.184} C_VEL
LIN {X 0,Y 178.487,Z 513.375,A -85,B 0,C 180,E1 -22618.197,E2 -22618.197} C_VEL
LIN {X 0,Y 178.477,Z 513.377,A -85,B 0,C 180,E1 -22620.791,E2 -22620.791} C_VEL
LIN {X 0,Y 178.496,Z 513.371,A -85,B 0,C 180,E1 -22624.224,E2 -22624.224} C_VEL
LIN {X 0,Y 178.419,Z 513.386,A -85,B 0,C 180,E1 -22629.068,E2 -22629.068} C_VEL
LIN {X 0,Y 178.413,Z 513.38,A -85,B 0,C 180,E1 -22632.041,E2 -22632.041} C_VEL
LIN {X 0,Y 178.401,Z 513.387,A -85,B 0,C 180,E1 -22635.162,E2 -22635.162} C_VEL
LIN {X 0,Y 178.514,Z 513.533,A -85,B 0,C 180,E1 -22638.953,E2 -22638.953} C_VEL
LIN {X 0,Y 181.981,Z 528.605,A -85,B 0,C 180,E1 -22643.724,E2 -22643.724} C_VEL
LIN {X 0,Y 185.589,Z 544.825,A -85,B 0,C 180,E1 -22648.621,E2 -22648.621} C_VEL
LIN {X 0,Y 184.741,Z 552.089,A -85,B 0,C 180,E1 -22650.611,E2 -22650.611} C_VEL
LIN {X 0,Y 186.069,Z 575.789,A -85,B 0,C 180,E1 -22652.3,E2 -22652.3} C_VEL
LIN {X 0,Y 187.037,Z 587.387,A -85,B 0,C 180,E1 -22653.13,E2 -22653.13} C_VEL
LIN {X 0,Y 183.313,Z 658.115,A -85,B 0,C 180,E1 -22658.05,E2 -22658.05} C_VEL
LIN {X 0,Y 182.51,Z 672.449,A -85,B 0,C 180,E1 -22659.281,E2 -22659.281} C_VEL
LIN {X 0,Y 181.384,Z 687.179,A -85,B 0,C 180,E1 -22661.065,E2 -22661.065} C_VEL
LIN {X 0,Y 180.161,Z 700.918,A -85,B 0,C 180,E1 -22663.28,E2 -22663.28} C_VEL
LIN {X 0,Y 179.112,Z 713.206,A -85,B 0,C 180,E1 -22665.804,E2 -22665.804} C_VEL
LIN {X 0,Y 178.088,Z 724.17,A -85,B 0,C 180,E1 -22668.62,E2 -22668.62} C_VEL
LIN {X 0,Y 177.429,Z 733.513,A -85,B 0,C 180,E1 -22671.587,E2 -22671.587} C_VEL
LIN {X 0,Y 176.954,Z 742.014,A -85,B 0,C 180,E1 -22674.879,E2 -22674.879} C_VEL
LIN {X 0,Y 176.727,Z 749.195,A -85,B 0,C 180,E1 -22678.291,E2 -22678.291} C_VEL
LIN {X 0,Y 176.613,Z 754.023,A -85,B 0,C 180,E1 -22681.14,E2 -22681.14} C_VEL
LIN {X 0,Y 176.675,Z 758.719,A -85,B 0,C 180,E1 -22684.563,E2 -22684.563} C_VEL
LIN {X 0,Y 177.199,Z 762.422,A -85,B 0,C 180,E1 -22687.979,E2 -22687.979} C_VEL
LIN {X 0,Y 178.363,Z 765.2,A -85,B 0,C 180,E1 -22691.362,E2 -22691.362} C_VEL
LIN {X 0,Y 180.839,Z 767.623,A -85,B 0,C 180,E1 -22695.786,E2 -22695.786} C_VEL
LIN {X 0,Y 184.517,Z 768.647,A -85,B 0,C 180,E1 -22700.047,E2 -22700.047} C_VEL
LIN {X 0,Y 186.742,Z 768.622,A -85,B 0,C 180,E1 -22702.108,E2 -22702.108} C_VEL
LIN {X 0,Y 192.359,Z 767.5,A -85,B 0,C 180,E1 -22706.004,E2 -22706.004} C_VEL
LIN {X 0,Y 199.019,Z 765.006,A -85,B 0,C 180,E1 -22709.629,E2 -22709.629} C_VEL
LIN {X 0,Y 204.665,Z 762.147,A -85,B 0,C 180,E1 -22712.158,E2 -22712.158} C_VEL
LIN {X 0,Y 212.954,Z 756.983,A -85,B 0,C 180,E1 -22715.278,E2 -22715.278} C_VEL
LIN {X 0,Y 219.724,Z 751.988,A -85,B 0,C 180,E1 -22717.425,E2 -22717.425} C_VEL
LIN {X 0,Y 229.416,Z 743.64,A -85,B 0,C 180,E1 -22720.04,E2 -22720.04} C_VEL
LIN {X 0,Y 238.08,Z 734.886,A -85,B 0,C 180,E1 -22722.031,E2 -22722.031} C_VEL
LIN {X 0,Y 246.108,Z 725.512,A -85,B 0,C 180,E1 -22723.608,E2 -22723.608} C_VEL
LIN {X 0,Y 246.964,Z 724.459,A -85,B 0,C 180,E1 -22723.763,E2 -22723.763} C_VEL
LIN {X 0,Y 247.824,Z 723.349,A -85,B 0,C 180,E1 -22724.335,E2 -22724.335} C_VEL
LIN {X 0,Y 239.487,Z 733.456,A -85,B 0,C 180,E1 -22725.816,E2 -22725.816} C_VEL
LIN {X 0,Y 231.345,Z 742.089,A -85,B 0,C 180,E1 -22727.473,E2 -22727.473} C_VEL
LIN {X 0,Y 222.451,Z 750.501,A -85,B 0,C 180,E1 -22729.634,E2 -22729.634} C_VEL
LIN {X 0,Y 214.569,Z 757.075,A -85,B 0,C 180,E1 -22731.875,E2 -22731.875} C_VEL
LIN {X 0,Y 210.724,Z 759.815,A -85,B 0,C 180,E1 -22732.841,E2 -22732.841} C_VEL
LIN {X 0,Y 200.244,Z 765.601,A -85,B 0,C 180,E1 -22734.801,E2 -22734.801} C_VEL
LIN {X 0,Y 194.627,Z 768.199,A -85,B 0,C 180,E1 -22736.201,E2 -22736.201} C_VEL
LIN {X 0,Y 192.335,Z 769.215,A -85,B 0,C 180,E1 -22737.087,E2 -22737.087} C_VEL
LIN {X 0,Y 185.713,Z 772.007,A -85,B 0,C 180,E1 -22740.53,E2 -22740.53} C_VEL
LIN {X 0,Y 179.96,Z 773.723,A -85,B 0,C 180,E1 -22744.559,E2 -22744.559} C_VEL
LIN {X 0,Y 175.397,Z 774.186,A -85,B 0,C 180,E1 -22748.862,E2 -22748.862} C_VEL
LIN {X 0,Y 172.123,Z 773.344,A -85,B 0,C 180,E1 -22753.392,E2 -22753.392} C_VEL
LIN {X 0,Y 170.377,Z 771.193,A -85,B 0,C 180,E1 -22758.098,E2 -22758.098} C_VEL
LIN {X 0,Y 169.84,Z 767.65,A -85,B 0,C 180,E1 -22762.869,E2 -22762.869} C_VEL
LIN {X 0,Y 170.105,Z 763.926,A -85,B 0,C 180,E1 -22766.447,E2 -22766.447} C_VEL
LIN {X 0,Y 170.401,Z 760.905,A -85,B 0,C 180,E1 -22768.819,E2 -22768.819} C_VEL
LIN {X 0,Y 169.807,Z 766.315,A -85,B 0,C 180,E1 -22773.559,E2 -22773.559} C_VEL
LIN {X 0,Y 169.594,Z 769.294,A -85,B 0,C 180,E1 -22777.142,E2 -22777.142} C_VEL
LIN {X 0,Y 170.193,Z 772.123,A -85,B 0,C 180,E1 -22781.916,E2 -22781.916} C_VEL
LIN {X 0,Y 171.887,Z 773.75,A -85,B 0,C 180,E1 -22786.632,E2 -22786.632} C_VEL
LIN {X 0,Y 175.037,Z 774.258,A -85,B 0,C 180,E1 -22791.184,E2 -22791.184} C_VEL
LIN {X 0,Y 180.178,Z 773.455,A -85,B 0,C 180,E1 -22796.216,E2 -22796.216} C_VEL
LIN {X 0,Y 184.939,Z 771.963,A -85,B 0,C 180,E1 -22799.606,E2 -22799.606} C_VEL
LIN {X 0,Y 191.562,Z 769.179,A -85,B 0,C 180,E1 -22803.389,E2 -22803.389} C_VEL
LIN {X 0,Y 199.373,Z 765.202,A -85,B 0,C 180,E1 -22806.817,E2 -22806.817} C_VEL
LIN {X 0,Y 208.105,Z 760.021,A -85,B 0,C 180,E1 -22809.916,E2 -22809.916} C_VEL
LIN {X 0,Y 217.708,Z 753.485,A -85,B 0,C 180,E1 -22812.681,E2 -22812.681} C_VEL
LIN {X 0,Y 228.062,Z 745.422,A -85,B 0,C 180,E1 -22815.136,E2 -22815.136} C_VEL
LIN {X 0,Y 236.397,Z 738.126,A -85,B 0,C 180,E1 -22816.789,E2 -22816.789} C_VEL
LIN {X 0,Y 237.995,Z 736.61,A -85,B 0,C 180,E1 -22817.22,E2 -22817.22} C_VEL
LIN {X 0,Y 228.387,Z 744.71,A -85,B 0,C 180,E1 -22819.163,E2 -22819.163} C_VEL
LIN {X 0,Y 219.352,Z 751.349,A -85,B 0,C 180,E1 -22821.334,E2 -22821.334} C_VEL
LIN {X 0,Y 209.668,Z 757.452,A -85,B 0,C 180,E1 -22824.084,E2 -22824.084} C_VEL
LIN {X 0,Y 202.974,Z 761.054,A -85,B 0,C 180,E1 -22826.358,E2 -22826.358} C_VEL
LIN {X 0,Y 194.875,Z 764.639,A -85,B 0,C 180,E1 -22829.675,E2 -22829.675} C_VEL
LIN {X 0,Y 187.822,Z 766.892,A -85,B 0,C 180,E1 -22833.319,E2 -22833.319} C_VEL
LIN {X 0,Y 181.766,Z 767.893,A -85,B 0,C 180,E1 -22837.254,E2 -22837.254} C_VEL
LIN {X 0,Y 176.813,Z 767.601,A -85,B 0,C 180,E1 -22841.459,E2 -22841.459} C_VEL
LIN {X 0,Y 173.314,Z 766.001,A -85,B 0,C 180,E1 -22845.918,E2 -22845.918} C_VEL
LIN {X 0,Y 170.879,Z 763.008,A -85,B 0,C 180,E1 -22850.531,E2 -22850.531} C_VEL
LIN {X 0,Y 169.779,Z 758.604,A -85,B 0,C 180,E1 -22855.251,E2 -22855.251} C_VEL
LIN {X 0,Y 169.549,Z 754.225,A -85,B 0,C 180,E1 -22858.812,E2 -22858.812} C_VEL
LIN {X 0,Y 169.485,Z 748.765,A -85,B 0,C 180,E1 -22862.376,E2 -22862.376} C_VEL
LIN {X 0,Y 169.782,Z 741.971,A -85,B 0,C 180,E1 -22865.941,E2 -22865.941} C_VEL
LIN {X 0,Y 170.228,Z 733.608,A -85,B 0,C 180,E1 -22869.505,E2 -22869.505} C_VEL
LIN {X 0,Y 171.074,Z 723.446,A -85,B 0,C 180,E1 -22873.059,E2 -22873.059} C_VEL
LIN {X 0,Y 171.897,Z 714.223,A -85,B 0,C 180,E1 -22875.716,E2 -22875.716} C_VEL
LIN {X 0,Y 173.285,Z 701.801,A -85,B 0,C 180,E1 -22878.626,E2 -22878.626} C_VEL
LIN {X 0,Y 174.627,Z 689.716,A -85,B 0,C 180,E1 -22880.927,E2 -22880.927} C_VEL
LIN {X 0,Y 175.914,Z 676.564,A -85,B 0,C 180,E1 -22882.917,E2 -22882.917} C_VEL
LIN {X 0,Y 177.214,Z 661.34,A -85,B 0,C 180,E1 -22884.685,E2 -22884.685} C_VEL
LIN {X 0,Y 178.76,Z 639.05,A -85,B 0,C 180,E1 -22886.486,E2 -22886.486} C_VEL
LIN {X 0,Y 182.361,Z 585.076,A -85,B 0,C 180,E1 -22890.404,E2 -22890.404} C_VEL
LIN {X 0,Y 179.757,Z 552.136,A -85,B 0,C 180,E1 -22893.027,E2 -22893.027} C_VEL
LIN {X 0,Y 179.357,Z 548.379,A -85,B 0,C 180,E1 -22893.333,E2 -22893.333} C_VEL
LIN {X 0,Y 176.444,Z 537.222,A -85,B 0,C 180,E1 -22894.42,E2 -22894.42} C_VEL
LIN {X 0,Y 174.216,Z 526.955,A -85,B 0,C 180,E1 -22899.135,E2 -22899.135} C_VEL
LIN {X 0,Y 171.997,Z 516.954,A -85,B 0,C 180,E1 -22903.999,E2 -22903.999} C_VEL
LIN {X 0,Y 171.345,Z 514.268,A -85,B 0,C 180,E1 -22905.417,E2 -22905.417} C_VEL
LIN {X 0,Y 171.359,Z 514.265,A -85,B 0,C 180,E1 -22911.192,E2 -22911.192} C_VEL
LIN {X 0,Y 171.4,Z 514.256,A -85,B 0,C 180,E1 -22915.092,E2 -22915.092} C_VEL
LIN {X 0,Y 171.451,Z 514.252,A -85,B 0,C 180,E1 -22920.534,E2 -22920.534} C_VEL
LIN {X 0,Y 171.459,Z 514.251,A -85,B 0,C 180,E1 -22925.802,E2 -22925.802} C_VEL
LIN {X 0,Y 171.581,Z 514.235,A -85,B 0,C 180,E1 -22930.872,E2 -22930.872} C_VEL
LIN {X 0,Y 171.611,Z 514.234,A -85,B 0,C 180,E1 -22935.776,E2 -22935.776} C_VEL
LIN {X 0,Y 171.912,Z 514.191,A -85,B 0,C 180,E1 -22940.588,E2 -22940.588} C_VEL
LIN {X 0,Y 171.83,Z 514.207,A -85,B 0,C 180,E1 -22945.308,E2 -22945.308} C_VEL
LIN {X 0,Y 172.337,Z 514.138,A -85,B 0,C 180,E1 -22950,E2 -22950} C_VEL
LIN {X 0,Y 171.828,Z 514.205,A -85,B 0,C 180,E1 -22954.692,E2 -22954.692} C_VEL
LIN {X 0,Y 171.912,Z 514.193,A -85,B 0,C 180,E1 -22959.412,E2 -22959.412} C_VEL
LIN {X 0,Y 171.614,Z 514.231,A -85,B 0,C 180,E1 -22964.224,E2 -22964.224} C_VEL
LIN {X 0,Y 171.559,Z 514.241,A -85,B 0,C 180,E1 -22969.575,E2 -22969.575} C_VEL
LIN {X 0,Y 171.469,Z 514.247,A -85,B 0,C 180,E1 -22975.616,E2 -22975.616} C_VEL
LIN {X 0,Y 171.44,Z 514.253,A -85,B 0,C 180,E1 -22980.585,E2 -22980.585} C_VEL
LIN {X 0,Y 171.407,Z 514.255,A -85,B 0,C 180,E1 -22985.032,E2 -22985.032} C_VEL
LIN {X 0,Y 171.381,Z 514.261,A -85,B 0,C 180,E1 -22988.817,E2 -22988.817} C_VEL
LIN {X 0,Y 171.331,Z 514.266,A -85,B 0,C 180,E1 -22994.214,E2 -22994.214} C_VEL
LIN {X 0,Y 171.408,Z 514.312,A -85,B 0,C 180,E1 -22998.435,E2 -22998.435} C_VEL
LIN {X 0,Y 174.967,Z 529.669,A -85,B 0,C 180,E1 -23003.452,E2 -23003.452} C_VEL
LIN {X 0,Y 178.596,Z 546.167,A -85,B 0,C 180,E1 -23008.573,E2 -23008.573} C_VEL
LIN {X 0,Y 177.724,Z 552.245,A -85,B 0,C 180,E1 -23010.273,E2 -23010.273} C_VEL
LIN {X 0,Y 179.085,Z 576.976,A -85,B 0,C 180,E1 -23012.126,E2 -23012.126} C_VEL
LIN {X 0,Y 179.95,Z 587.569,A -85,B 0,C 180,E1 -23012.92,E2 -23012.92} C_VEL
LIN {X 0,Y 176.027,Z 662.268,A -85,B 0,C 180,E1 -23018.404,E2 -23018.404} C_VEL
LIN {X 0,Y 175.043,Z 677.158,A -85,B 0,C 180,E1 -23019.892,E2 -23019.892} C_VEL
LIN {X 0,Y 173.964,Z 690.725,A -85,B 0,C 180,E1 -23021.754,E2 -23021.754} C_VEL
LIN {X 0,Y 172.838,Z 703.638,A -85,B 0,C 180,E1 -23024.07,E2 -23024.07} C_VEL
LIN {X 0,Y 171.805,Z 715.258,A -85,B 0,C 180,E1 -23026.697,E2 -23026.697} C_VEL
LIN {X 0,Y 170.995,Z 724.851,A -85,B 0,C 180,E1 -23029.342,E2 -23029.342} C_VEL
LIN {X 0,Y 170.354,Z 734.085,A -85,B 0,C 180,E1 -23032.429,E2 -23032.429} C_VEL
LIN {X 0,Y 169.963,Z 741.156,A -85,B 0,C 180,E1 -23035.256,E2 -23035.256} C_VEL
LIN {X 0,Y 169.767,Z 748.422,A -85,B 0,C 180,E1 -23038.814,E2 -23038.814} C_VEL
LIN {X 0,Y 169.678,Z 754.27,A -85,B 0,C 180,E1 -23042.374,E2 -23042.374} C_VEL
LIN {X 0,Y 169.849,Z 759.254,A -85,B 0,C 180,E1 -23046.225,E2 -23046.225} C_VEL
LIN {X 0,Y 170.61,Z 762.591,A -85,B 0,C 180,E1 -23049.484,E2 -23049.484} C_VEL
LIN {X 0,Y 172.53,Z 766.138,A -85,B 0,C 180,E1 -23054.147,E2 -23054.147} C_VEL
LIN {X 0,Y 175.837,Z 768.251,A -85,B 0,C 180,E1 -23058.648,E2 -23058.648} C_VEL
LIN {X 0,Y 180.199,Z 768.974,A -85,B 0,C 180,E1 -23062.955,E2 -23062.955} C_VEL
LIN {X 0,Y 186.071,Z 768.343,A -85,B 0,C 180,E1 -23066.952,E2 -23066.952} C_VEL
LIN {X 0,Y 192.99,Z 766.344,A -85,B 0,C 180,E1 -23070.652,E2 -23070.652} C_VEL
LIN {X 0,Y 200.909,Z 762.873,A -85,B 0,C 180,E1 -23074.035,E2 -23074.035} C_VEL
LIN {X 0,Y 209.722,Z 757.929,A -85,B 0,C 180,E1 -23077.099,E2 -23077.099} C_VEL
LIN {X 0,Y 216.88,Z 753.122,A -85,B 0,C 180,E1 -23079.19,E2 -23079.19} C_VEL
LIN {X 0,Y 226.111,Z 745.872,A -85,B 0,C 180,E1 -23081.515,E2 -23081.515} C_VEL
LIN {X 0,Y 235.072,Z 737.646,A -85,B 0,C 180,E1 -23083.443,E2 -23083.443} C_VEL
LIN {X 0,Y 236.581,Z 736.169,A -85,B 0,C 180,E1 -23083.733,E2 -23083.733} C_VEL
LIN {X 0,Y 237.307,Z 735.438,A -85,B 0,C 180,E1 -23084.262,E2 -23084.262} C_VEL
LIN {X 0,Y 227.872,Z 744.591,A -85,B 0,C 180,E1 -23086.057,E2 -23086.057} C_VEL
LIN {X 0,Y 218.623,Z 752.395,A -85,B 0,C 180,E1 -23088.161,E2 -23088.161} C_VEL
LIN {X 0,Y 209.938,Z 758.834,A -85,B 0,C 180,E1 -23090.502,E2 -23090.502} C_VEL
LIN {X 0,Y 200.868,Z 764.68,A -85,B 0,C 180,E1 -23093.502,E2 -23093.502} C_VEL
LIN {X 0,Y 192.335,Z 769.215,A -85,B 0,C 180,E1 -23097.087,E2 -23097.087} C_VEL
LIN {X 0,Y 188.802,Z 770.661,A -85,B 0,C 180,E1 -23098.457,E2 -23098.457} C_VEL
LIN {X 0,Y 181.803,Z 772.528,A -85,B 0,C 180,E1 -23100.557,E2 -23100.557} C_VEL
LIN {X 0,Y 175.197,Z 773.572,A -85,B 0,C 180,E1 -23102.874,E2 -23102.874} C_VEL
LIN {X 0,Y 172.352,Z 773.759,A -85,B 0,C 180,E1 -23104.56,E2 -23104.56} C_VEL
LIN {X 0,Y 168.812,Z 773.702,A -85,B 0,C 180,E1 -23107.995,E2 -23107.995} C_VEL
LIN {X 0,Y 165.375,Z 772.478,A -85,B 0,C 180,E1 -23112.694,E2 -23112.694} C_VEL
LIN {X 0,Y 163.506,Z 769.997,A -85,B 0,C 180,E1 -23117.589,E2 -23117.589} C_VEL
LIN {X 0,Y 162.981,Z 765.983,A -85,B 0,C 180,E1 -23122.658,E2 -23122.658} C_VEL
LIN {X 0,Y 163.263,Z 762.079,A -85,B 0,C 180,E1 -23126.298,E2 -23126.298} C_VEL
LIN {X 0,Y 163.584,Z 758.929,A -85,B 0,C 180,E1 -23128.769,E2 -23128.769} C_VEL
LIN {X 0,Y 162.917,Z 764.69,A -85,B 0,C 180,E1 -23133.71,E2 -23133.71} C_VEL
LIN {X 0,Y 162.683,Z 767.945,A -85,B 0,C 180,E1 -23137.447,E2 -23137.447} C_VEL
LIN {X 0,Y 163.303,Z 771.072,A -85,B 0,C 180,E1 -23142.426,E2 -23142.426} C_VEL
LIN {X 0,Y 165.101,Z 773.004,A -85,B 0,C 180,E1 -23147.336,E2 -23147.336} C_VEL
LIN {X 0,Y 168.417,Z 773.849,A -85,B 0,C 180,E1 -23152.06,E2 -23152.06} C_VEL
LIN {X 0,Y 173.417,Z 773.54,A -85,B 0,C 180,E1 -23156.927,E2 -23156.927} C_VEL
LIN {X 0,Y 178.811,Z 772.287,A -85,B 0,C 180,E1 -23160.728,E2 -23160.728} C_VEL
LIN {X 0,Y 185.713,Z 769.92,A -85,B 0,C 180,E1 -23164.587,E2 -23164.587} C_VEL
LIN {X 0,Y 193.839,Z 766.446,A -85,B 0,C 180,E1 -23168.052,E2 -23168.052} C_VEL
LIN {X 0,Y 202.858,Z 761.786,A -85,B 0,C 180,E1 -23171.167,E2 -23171.167} C_VEL
LIN {X 0,Y 212.757,Z 755.832,A -85,B 0,C 180,E1 -23173.924,E2 -23173.924} C_VEL
LIN {X 0,Y 223.386,Z 748.525,A -85,B 0,C 180,E1 -23176.354,E2 -23176.354} C_VEL
LIN {X 0,Y 227.579,Z 745.297,A -85,B 0,C 180,E1 -23177.204,E2 -23177.204} C_VEL
LIN {X 0,Y 219.379,Z 751.037,A -85,B 0,C 180,E1 -23178.948,E2 -23178.948} C_VEL
LIN {X 0,Y 209.057,Z 757.214,A -85,B 0,C 180,E1 -23181.543,E2 -23181.543} C_VEL
LIN {X 0,Y 199.501,Z 761.951,A -85,B 0,C 180,E1 -23184.461,E2 -23184.461} C_VEL
LIN {X 0,Y 192.983,Z 764.615,A -85,B 0,C 180,E1 -23186.889,E2 -23186.889} C_VEL
LIN {X 0,Y 185.06,Z 767.031,A -85,B 0,C 180,E1 -23190.416,E2 -23190.416} C_VEL
LIN {X 0,Y 178.269,Z 768.179,A -85,B 0,C 180,E1 -23194.3,E2 -23194.3} C_VEL
LIN {X 0,Y 172.471,Z 768.095,A -85,B 0,C 180,E1 -23198.485,E2 -23198.485} C_VEL
LIN {X 0,Y 168.179,Z 766.732,A -85,B 0,C 180,E1 -23202.991,E2 -23202.991} C_VEL
LIN {X 0,Y 165.06,Z 764.087,A -85,B 0,C 180,E1 -23207.708,E2 -23207.708} C_VEL
LIN {X 0,Y 163.19,Z 760.04,A -85,B 0,C 180,E1 -23212.577,E2 -23212.577} C_VEL
LIN {X 0,Y 162.672,Z 756.025,A -85,B 0,C 180,E1 -23216.284,E2 -23216.284} C_VEL
LIN {X 0,Y 162.544,Z 750.965,A -85,B 0,C 180,E1 -23220,E2 -23220} C_VEL
LIN {X 0,Y 162.64,Z 743.584,A -85,B 0,C 180,E1 -23224.332,E2 -23224.332} C_VEL
LIN {X 0,Y 163.082,Z 735.704,A -85,B 0,C 180,E1 -23228.051,E2 -23228.051} C_VEL
LIN {X 0,Y 163.7,Z 725.863,A -85,B 0,C 180,E1 -23231.767,E2 -23231.767} C_VEL
LIN {X 0,Y 164.681,Z 716.062,A -85,B 0,C 180,E1 -23234.836,E2 -23234.836} C_VEL
LIN {X 0,Y 165.854,Z 704.187,A -85,B 0,C 180,E1 -23237.892,E2 -23237.892} C_VEL
LIN {X 0,Y 167.327,Z 691.122,A -85,B 0,C 180,E1 -23240.595,E2 -23240.595} C_VEL
LIN {X 0,Y 168.677,Z 677.879,A -85,B 0,C 180,E1 -23242.747,E2 -23242.747} C_VEL
LIN {X 0,Y 169.97,Z 663.078,A -85,B 0,C 180,E1 -23244.587,E2 -23244.587} C_VEL
LIN {X 0,Y 171.215,Z 646.015,A -85,B 0,C 180,E1 -23246.103,E2 -23246.103} C_VEL
LIN {X 0,Y 175.35,Z 585.636,A -85,B 0,C 180,E1 -23250.732,E2 -23250.732} C_VEL
LIN {X 0,Y 172.806,Z 552.175,A -85,B 0,C 180,E1 -23253.501,E2 -23253.501} C_VEL
LIN {X 0,Y 171.688,Z 546.823,A -85,B 0,C 180,E1 -23254.003,E2 -23254.003} C_VEL
LIN {X 0,Y 169.201,Z 537.123,A -85,B 0,C 180,E1 -23255.002,E2 -23255.002} C_VEL
LIN {X 0,Y 166.975,Z 527.05,A -85,B 0,C 180,E1 -23259.835,E2 -23259.835} C_VEL
LIN {X 0,Y 164.599,Z 516.502,A -85,B 0,C 180,E1 -23265.211,E2 -23265.211} C_VEL
LIN {X 0,Y 164.279,Z 515.149,A -85,B 0,C 180,E1 -23265.959,E2 -23265.959} C_VEL
LIN {X 0,Y 164.296,Z 515.144,A -85,B 0,C 180,E1 -23270.352,E2 -23270.352} C_VEL
LIN {X 0,Y 164.331,Z 515.136,A -85,B 0,C 180,E1 -23276.222,E2 -23276.222} C_VEL
LIN {X 0,Y 164.407,Z 515.13,A -85,B 0,C 180,E1 -23279.138,E2 -23279.138} C_VEL
LIN {X 0,Y 164.418,Z 515.123,A -85,B 0,C 180,E1 -23284.694,E2 -23284.694} C_VEL
LIN {X 0,Y 164.486,Z 515.119,A -85,B 0,C 180,E1 -23290.051,E2 -23290.051} C_VEL
LIN {X 0,Y 164.555,Z 515.11,A -85,B 0,C 180,E1 -23295.152,E2 -23295.152} C_VEL
LIN {X 0,Y 164.854,Z 515.07,A -85,B 0,C 180,E1 -23300.181,E2 -23300.181} C_VEL
LIN {X 0,Y 164.78,Z 515.084,A -85,B 0,C 180,E1 -23305.106,E2 -23305.106} C_VEL
LIN {X 0,Y 165.299,Z 515.015,A -85,B 0,C 180,E1 -23310,E2 -23310} C_VEL
LIN {X 0,Y 164.779,Z 515.084,A -85,B 0,C 180,E1 -23314.893,E2 -23314.893} C_VEL
LIN {X 0,Y 164.854,Z 515.074,A -85,B 0,C 180,E1 -23319.818,E2 -23319.818} C_VEL
LIN {X 0,Y 164.56,Z 515.11,A -85,B 0,C 180,E1 -23324.847,E2 -23324.847} C_VEL
LIN {X 0,Y 164.476,Z 515.121,A -85,B 0,C 180,E1 -23329.989,E2 -23329.989} C_VEL
LIN {X 0,Y 164.394,Z 515.128,A -85,B 0,C 180,E1 -23336.133,E2 -23336.133} C_VEL
LIN {X 0,Y 164.375,Z 515.135,A -85,B 0,C 180,E1 -23341.227,E2 -23341.227} C_VEL
LIN {X 0,Y 164.314,Z 515.141,A -85,B 0,C 180,E1 -23346.784,E2 -23346.784} C_VEL
LIN {X 0,Y 164.301,Z 515.141,A -85,B 0,C 180,E1 -23349.913,E2 -23349.913} C_VEL
LIN {X 0,Y 164.28,Z 515.143,A -85,B 0,C 180,E1 -23353.342,E2 -23353.342} C_VEL
LIN {X 0,Y 164.346,Z 515.154,A -85,B 0,C 180,E1 -23357.942,E2 -23357.942} C_VEL
LIN {X 0,Y 167.689,Z 529.505,A -85,B 0,C 180,E1 -23362.779,E2 -23362.779} C_VEL
LIN {X 0,Y 171.324,Z 546.005,A -85,B 0,C 180,E1 -23368.073,E2 -23368.073} C_VEL
LIN {X 0,Y 171.513,Z 547.1,A -85,B 0,C 180,E1 -23368.412,E2 -23368.412} C_VEL
LIN {X 0,Y 170.696,Z 552.482,A -85,B 0,C 180,E1 -23369.962,E2 -23369.962} C_VEL
LIN {X 0,Y 172.038,Z 577.366,A -85,B 0,C 180,E1 -23371.906,E2 -23371.906} C_VEL
LIN {X 0,Y 172.895,Z 587.587,A -85,B 0,C 180,E1 -23372.705,E2 -23372.705} C_VEL
LIN {X 0,Y 168.967,Z 661.585,A -85,B 0,C 180,E1 -23378.417,E2 -23378.417} C_VEL
LIN {X 0,Y 167.998,Z 676.477,A -85,B 0,C 180,E1 -23379.97,E2 -23379.97} C_VEL
LIN {X 0,Y 167.086,Z 688.244,A -85,B 0,C 180,E1 -23381.611,E2 -23381.611} C_VEL
LIN {X 0,Y 165.922,Z 701.64,A -85,B 0,C 180,E1 -23384.019,E2 -23384.019} C_VEL
LIN {X 0,Y 164.854,Z 713.645,A -85,B 0,C 180,E1 -23386.753,E2 -23386.753} C_VEL
LIN {X 0,Y 164.041,Z 723.517,A -85,B 0,C 180,E1 -23389.509,E2 -23389.509} C_VEL
LIN {X 0,Y 163.425,Z 732.617,A -85,B 0,C 180,E1 -23392.587,E2 -23392.587} C_VEL
LIN {X 0,Y 163.028,Z 740.146,A -85,B 0,C 180,E1 -23395.673,E2 -23395.673} C_VEL
LIN {X 0,Y 162.822,Z 747.588,A -85,B 0,C 180,E1 -23399.382,E2 -23399.382} C_VEL
LIN {X 0,Y 162.745,Z 752.675,A -85,B 0,C 180,E1 -23402.475,E2 -23402.475} C_VEL
LIN {X 0,Y 163.033,Z 759.035,A -85,B 0,C 180,E1 -23407.431,E2 -23407.431} C_VEL
LIN {X 0,Y 164.074,Z 762.709,A -85,B 0,C 180,E1 -23411.114,E2 -23411.114} C_VEL
LIN {X 0,Y 165.676,Z 765.528,A -85,B 0,C 180,E1 -23414.745,E2 -23414.745} C_VEL
LIN {X 0,Y 169.134,Z 768.029,A -85,B 0,C 180,E1 -23419.416,E2 -23419.416} C_VEL
LIN {X 0,Y 173.703,Z 769.205,A -85,B 0,C 180,E1 -23423.866,E2 -23423.866} C_VEL
LIN {X 0,Y 179.803,Z 769.049,A -85,B 0,C 180,E1 -23427.973,E2 -23427.973} C_VEL
LIN {X 0,Y 186.998,Z 767.519,A -85,B 0,C 180,E1 -23431.747,E2 -23431.747} C_VEL
LIN {X 0,Y 195.212,Z 764.624,A -85,B 0,C 180,E1 -23435.172,E2 -23435.172} C_VEL
LIN {X 0,Y 204.332,Z 760.306,A -85,B 0,C 180,E1 -23438.251,E2 -23438.251} C_VEL
LIN {X 0,Y 214.275,Z 754.333,A -85,B 0,C 180,E1 -23440.994,E2 -23440.994} C_VEL
LIN {X 0,Y 223.519,Z 747.699,A -85,B 0,C 180,E1 -23443.147,E2 -23443.147} C_VEL
LIN {X 0,Y 226.134,Z 745.634,A -85,B 0,C 180,E1 -23443.704,E2 -23443.704} C_VEL
LIN {X 0,Y 226.739,Z 745.171,A -85,B 0,C 180,E1 -23444.176,E2 -23444.176} C_VEL
LIN {X 0,Y 217.671,Z 752.315,A -85,B 0,C 180,E1 -23446.038,E2 -23446.038} C_VEL
LIN {X 0,Y 209.726,Z 757.823,A -85,B 0,C 180,E1 -23447.917,E2 -23447.917} C_VEL
LIN {X 0,Y 202.277,Z 762.436,A -85,B 0,C 180,E1 -23450.001,E2 -23450.001} C_VEL
LIN {X 0,Y 193.139,Z 767.232,A -85,B 0,C 180,E1 -23453.101,E2 -23453.101} C_VEL
LIN {X 0,Y 186.544,Z 770.102,A -85,B 0,C 180,E1 -23455.883,E2 -23455.883} C_VEL
LIN {X 0,Y 179.593,Z 772.433,A -85,B 0,C 180,E1 -23459.421,E2 -23459.421} C_VEL
LIN {X 0,Y 173.573,Z 773.682,A -85,B 0,C 180,E1 -23463.552,E2 -23463.552} C_VEL
LIN {X 0,Y 172.352,Z 773.759,A -85,B 0,C 180,E1 -23464.56,E2 -23464.56} C_VEL
LIN {X 0,Y 169.709,Z 773.822,A -85,B 0,C 180,E1 -23466.328,E2 -23466.328} C_VEL
LIN {X 0,Y 164.194,Z 773.073,A -85,B 0,C 180,E1 -23469.14,E2 -23469.14} C_VEL
LIN {X 0,Y 159.274,Z 771.532,A -85,B 0,C 180,E1 -23472.135,E2 -23472.135} C_VEL
LIN {X 0,Y 157.63,Z 770.346,A -85,B 0,C 180,E1 -23474.147,E2 -23474.147} C_VEL
LIN {X 0,Y 156.248,Z 766.669,A -85,B 0,C 180,E1 -23479.635,E2 -23479.635} C_VEL
LIN {X 0,Y 156.322,Z 761.59,A -85,B 0,C 180,E1 -23484.841,E2 -23484.841} C_VEL
LIN {X 0,Y 156.84,Z 756.74,A -85,B 0,C 180,E1 -23488.636,E2 -23488.636} C_VEL
LIN {X 0,Y 156.179,Z 761.605,A -85,B 0,C 180,E1 -23492.579,E2 -23492.579} C_VEL
LIN {X 0,Y 155.813,Z 765.868,A -85,B 0,C 180,E1 -23497.106,E2 -23497.106} C_VEL
LIN {X 0,Y 156.466,Z 769.841,A -85,B 0,C 180,E1 -23502.979,E2 -23502.979} C_VEL
LIN {X 0,Y 158.362,Z 772.089,A -85,B 0,C 180,E1 -23508.099,E2 -23508.099} C_VEL
LIN {X 0,Y 161.85,Z 773.288,A -85,B 0,C 180,E1 -23513.005,E2 -23513.005} C_VEL
LIN {X 0,Y 166.61,Z 773.431,A -85,B 0,C 180,E1 -23517.646,E2 -23517.646} C_VEL
LIN {X 0,Y 172.736,Z 772.515,A -85,B 0,C 180,E1 -23521.933,E2 -23521.933} C_VEL
LIN {X 0,Y 179.953,Z 770.566,A -85,B 0,C 180,E1 -23525.861,E2 -23525.861} C_VEL
LIN {X 0,Y 188.366,Z 767.537,A -85,B 0,C 180,E1 -23529.367,E2 -23529.367} C_VEL
LIN {X 0,Y 197.697,Z 763.426,A -85,B 0,C 180,E1 -23532.489,E2 -23532.489} C_VEL
LIN {X 0,Y 207.899,Z 758.085,A -85,B 0,C 180,E1 -23535.227,E2 -23535.227} C_VEL
LIN {X 0,Y 216.07,Z 753.166,A -85,B 0,C 180,E1 -23537.077,E2 -23537.077} C_VEL
LIN {X 0,Y 215.37,Z 753.563,A -85,B 0,C 180,E1 -23537.548,E2 -23537.548} C_VEL
LIN {X 0,Y 206.357,Z 758.412,A -85,B 0,C 180,E1 -23539.677,E2 -23539.677} C_VEL
LIN {X 0,Y 196.321,Z 762.925,A -85,B 0,C 180,E1 -23542.513,E2 -23542.513} C_VEL
LIN {X 0,Y 186.692,Z 766.214,A -85,B 0,C 180,E1 -23545.914,E2 -23545.914} C_VEL
LIN {X 0,Y 178.99,Z 767.992,A -85,B 0,C 180,E1 -23549.307,E2 -23549.307} C_VEL
LIN {X 0,Y 171.915,Z 768.691,A -85,B 0,C 180,E1 -23553.276,E2 -23553.276} C_VEL
LIN {X 0,Y 165.889,Z 768.159,A -85,B 0,C 180,E1 -23557.586,E2 -23557.586} C_VEL
LIN {X 0,Y 161.421,Z 766.394,A -85,B 0,C 180,E1 -23562.256,E2 -23562.256} C_VEL
LIN {X 0,Y 158.188,Z 763.328,A -85,B 0,C 180,E1 -23567.165,E2 -23567.165} C_VEL
LIN {X 0,Y 156.244,Z 758.904,A -85,B 0,C 180,E1 -23572.245,E2 -23572.245} C_VEL
LIN {X 0,Y 155.727,Z 754.586,A -85,B 0,C 180,E1 -23576.118,E2 -23576.118} C_VEL
LIN {X 0,Y 155.59,Z 749.291,A -85,B 0,C 180,E1 -23580,E2 -23580} C_VEL
LIN {X 0,Y 155.71,Z 742.658,A -85,B 0,C 180,E1 -23583.882,E2 -23583.882} C_VEL
LIN {X 0,Y 156.207,Z 733.599,A -85,B 0,C 180,E1 -23588.181,E2 -23588.181} C_VEL
LIN {X 0,Y 156.728,Z 724.661,A -85,B 0,C 180,E1 -23591.642,E2 -23591.642} C_VEL
LIN {X 0,Y 157.705,Z 714.626,A -85,B 0,C 180,E1 -23594.847,E2 -23594.847} C_VEL
LIN {X 0,Y 158.932,Z 702.353,A -85,B 0,C 180,E1 -23598.032,E2 -23598.032} C_VEL
LIN {X 0,Y 160.266,Z 690.53,A -85,B 0,C 180,E1 -23600.537,E2 -23600.537} C_VEL
LIN {X 0,Y 161.578,Z 677.78,A -85,B 0,C 180,E1 -23602.707,E2 -23602.707} C_VEL
LIN {X 0,Y 162.873,Z 662.995,A -85,B 0,C 180,E1 -23604.654,E2 -23604.654} C_VEL
LIN {X 0,Y 164.158,Z 645.692,A -85,B 0,C 180,E1 -23606.285,E2 -23606.285} C_VEL
LIN {X 0,Y 168.293,Z 585.96,A -85,B 0,C 180,E1 -23611.076,E2 -23611.076} C_VEL
LIN {X 0,Y 165.696,Z 551.618,A -85,B 0,C 180,E1 -23614.061,E2 -23614.061} C_VEL
LIN {X 0,Y 161.908,Z 537.032,A -85,B 0,C 180,E1 -23615.609,E2 -23615.609} C_VEL
LIN {X 0,Y 159.698,Z 527.06,A -85,B 0,C 180,E1 -23620.611,E2 -23620.611} C_VEL
LIN {X 0,Y 157.627,Z 517.829,A -85,B 0,C 180,E1 -23625.511,E2 -23625.511} C_VEL
LIN {X 0,Y 157.237,Z 516.025,A -85,B 0,C 180,E1 -23626.548,E2 -23626.548} C_VEL
LIN {X 0,Y 157.207,Z 516.028,A -85,B 0,C 180,E1 -23631.253,E2 -23631.253} C_VEL
LIN {X 0,Y 157.28,Z 516.014,A -85,B 0,C 180,E1 -23634.486,E2 -23634.486} C_VEL
LIN {X 0,Y 157.303,Z 516.015,A -85,B 0,C 180,E1 -23638.091,E2 -23638.091} C_VEL
LIN {X 0,Y 157.324,Z 516.009,A -85,B 0,C 180,E1 -23643.466,E2 -23643.466} C_VEL
LIN {X 0,Y 157.395,Z 516.004,A -85,B 0,C 180,E1 -23649.667,E2 -23649.667} C_VEL
LIN {X 0,Y 157.48,Z 515.99,A -85,B 0,C 180,E1 -23654.468,E2 -23654.468} C_VEL
LIN {X 0,Y 157.774,Z 515.953,A -85,B 0,C 180,E1 -23659.736,E2 -23659.736} C_VEL
LIN {X 0,Y 157.826,Z 515.946,A -85,B 0,C 180,E1 -23662.323,E2 -23662.323} C_VEL
LIN {X 0,Y 158.261,Z 515.892,A -85,B 0,C 180,E1 -23670,E2 -23670} C_VEL
LIN {X 0,Y 157.826,Z 515.945,A -85,B 0,C 180,E1 -23677.677,E2 -23677.677} C_VEL
LIN {X 0,Y 157.707,Z 515.965,A -85,B 0,C 180,E1 -23681.362,E2 -23681.362} C_VEL
LIN {X 0,Y 157.487,Z 515.989,A -85,B 0,C 180,E1 -23685.531,E2 -23685.531} C_VEL
LIN {X 0,Y 157.372,Z 516.007,A -85,B 0,C 180,E1 -23690.932,E2 -23690.932} C_VEL
LIN {X 0,Y 157.315,Z 516.01,A -85,B 0,C 180,E1 -23696.684,E2 -23696.684} C_VEL
LIN {X 0,Y 157.278,Z 516.015,A -85,B 0,C 180,E1 -23702.427,E2 -23702.427} C_VEL
LIN {X 0,Y 157.283,Z 516.016,A -85,B 0,C 180,E1 -23706.457,E2 -23706.457} C_VEL
LIN {X 0,Y 157.214,Z 516.02,A -85,B 0,C 180,E1 -23712.11,E2 -23712.11} C_VEL
LIN {X 0,Y 157.318,Z 516.165,A -85,B 0,C 180,E1 -23717.499,E2 -23717.499} C_VEL
LIN {X 0,Y 160.893,Z 531.583,A -85,B 0,C 180,E1 -23722.86,E2 -23722.86} C_VEL
LIN {X 0,Y 164.371,Z 547.376,A -85,B 0,C 180,E1 -23728.056,E2 -23728.056} C_VEL
LIN {X 0,Y 163.672,Z 552.56,A -85,B 0,C 180,E1 -23729.61,E2 -23729.61} C_VEL
LIN {X 0,Y 164.965,Z 577.562,A -85,B 0,C 180,E1 -23731.653,E2 -23731.653} C_VEL
LIN {X 0,Y 165.796,Z 588.378,A -85,B 0,C 180,E1 -23732.539,E2 -23732.539} C_VEL
LIN {X 0,Y 161.994,Z 658.357,A -85,B 0,C 180,E1 -23738.277,E2 -23738.277} C_VEL
LIN {X 0,Y 161.158,Z 673.074,A -85,B 0,C 180,E1 -23739.748,E2 -23739.748} C_VEL
LIN {X 0,Y 160.056,Z 687.496,A -85,B 0,C 180,E1 -23741.769,E2 -23741.769} C_VEL
LIN {X 0,Y 158.898,Z 701.088,A -85,B 0,C 180,E1 -23744.282,E2 -23744.282} C_VEL
LIN {X 0,Y 157.923,Z 711.956,A -85,B 0,C 180,E1 -23746.816,E2 -23746.816} C_VEL
LIN {X 0,Y 157.03,Z 723.404,A -85,B 0,C 180,E1 -23750.149,E2 -23750.149} C_VEL
LIN {X 0,Y 156.42,Z 733.052,A -85,B 0,C 180,E1 -23753.585,E2 -23753.585} C_VEL
LIN {X 0,Y 156.058,Z 741.76,A -85,B 0,C 180,E1 -23757.419,E2 -23757.419} C_VEL
LIN {X 0,Y 155.909,Z 748.801,A -85,B 0,C 180,E1 -23761.292,E2 -23761.292} C_VEL
LIN {X 0,Y 155.877,Z 754.499,A -85,B 0,C 180,E1 -23765.174,E2 -23765.174} C_VEL
LIN {X 0,Y 156.799,Z 760.435,A -85,B 0,C 180,E1 -23770.328,E2 -23770.328} C_VEL
LIN {X 0,Y 158.87,Z 764.737,A -85,B 0,C 180,E1 -23775.392,E2 -23775.392} C_VEL
LIN {X 0,Y 162.469,Z 767.684,A -85,B 0,C 180,E1 -23780.247,E2 -23780.247} C_VEL
LIN {X 0,Y 167.258,Z 769.295,A -85,B 0,C 180,E1 -23784.847,E2 -23784.847} C_VEL
LIN {X 0,Y 173.59,Z 769.585,A -85,B 0,C 180,E1 -23789.067,E2 -23789.067} C_VEL
LIN {X 0,Y 181.076,Z 768.552,A -85,B 0,C 180,E1 -23792.914,E2 -23792.914} C_VEL
LIN {X 0,Y 189.582,Z 766.201,A -85,B 0,C 180,E1 -23796.38,E2 -23796.38} C_VEL
LIN {X 0,Y 199.001,Z 762.477,A -85,B 0,C 180,E1 -23799.472,E2 -23799.472} C_VEL
LIN {X 0,Y 209.235,Z 757.206,A -85,B 0,C 180,E1 -23802.205,E2 -23802.205} C_VEL
LIN {X 0,Y 214.627,Z 753.971,A -85,B 0,C 180,E1 -23803.444,E2 -23803.444} C_VEL
LIN {X 0,Y 215.621,Z 753.402,A -85,B 0,C 180,E1 -23804.186,E2 -23804.186} C_VEL
LIN {X 0,Y 204.689,Z 760.159,A -85,B 0,C 180,E1 -23806.631,E2 -23806.631} C_VEL
LIN {X 0,Y 194.58,Z 765.406,A -85,B 0,C 180,E1 -23809.448,E2 -23809.448} C_VEL
LIN {X 0,Y 185.428,Z 769.279,A -85,B 0,C 180,E1 -23812.668,E2 -23812.668} C_VEL
LIN {X 0,Y 177.247,Z 771.878,A -85,B 0,C 180,E1 -23816.281,E2 -23816.281} C_VEL
LIN {X 0,Y 170.198,Z 773.257,A -85,B 0,C 180,E1 -23820.296,E2 -23820.296} C_VEL
LIN {X 0,Y 164.572,Z 773.44,A -85,B 0,C 180,E1 -23824.72,E2 -23824.72} C_VEL
LIN {X 0,Y 160.286,Z 772.42,A -85,B 0,C 180,E1 -23829.465,E2 -23829.465} C_VEL
LIN {X 0,Y 157.63,Z 770.346,A -85,B 0,C 180,E1 -23834.147,E2 -23834.147} C_VEL
LIN {X 0,Y 156.272,Z 769.005,A -85,B 0,C 180,E1 -23836.189,E2 -23836.189} C_VEL
LIN {X 0,Y 152.897,Z 765.803,A -85,B 0,C 180,E1 -23839.437,E2 -23839.437} C_VEL
LIN {X 0,Y 150.057,Z 761.839,A -85,B 0,C 180,E1 -23842.725,E2 -23842.725} C_VEL
LIN {X 0,Y 149.586,Z 759.304,A -85,B 0,C 180,E1 -23844.774,E2 -23844.774} C_VEL
LIN {X 0,Y 150.155,Z 754.454,A -85,B 0,C 180,E1 -23848.492,E2 -23848.492} C_VEL
LIN {X 0,Y 149.258,Z 761.044,A -85,B 0,C 180,E1 -23854.05,E2 -23854.05} C_VEL
LIN {X 0,Y 148.972,Z 765.793,A -85,B 0,C 180,E1 -23859.504,E2 -23859.504} C_VEL
LIN {X 0,Y 149.668,Z 768.483,A -85,B 0,C 180,E1 -23863.579,E2 -23863.579} C_VEL
LIN {X 0,Y 151.689,Z 771.053,A -85,B 0,C 180,E1 -23868.925,E2 -23868.925} C_VEL
LIN {X 0,Y 155.355,Z 772.575,A -85,B 0,C 180,E1 -23874.026,E2 -23874.026} C_VEL
LIN {X 0,Y 160.349,Z 773.075,A -85,B 0,C 180,E1 -23878.825,E2 -23878.825} C_VEL
LIN {X 0,Y 166.748,Z 772.58,A -85,B 0,C 180,E1 -23883.225,E2 -23883.225} C_VEL
LIN {X 0,Y 174.271,Z 771.078,A -85,B 0,C 180,E1 -23887.223,E2 -23887.223} C_VEL
LIN {X 0,Y 182.997,Z 768.528,A -85,B 0,C 180,E1 -23890.76,E2 -23890.76} C_VEL
LIN {X 0,Y 192.632,Z 764.901,A -85,B 0,C 180,E1 -23893.884,E2 -23893.884} C_VEL
LIN {X 0,Y 203.108,Z 760.141,A -85,B 0,C 180,E1 -23896.607,E2 -23896.607} C_VEL
LIN {X 0,Y 205.402,Z 758.983,A -85,B 0,C 180,E1 -23897.126,E2 -23897.126} C_VEL
LIN {X 0,Y 204.695,Z 759.299,A -85,B 0,C 180,E1 -23897.574,E2 -23897.574} C_VEL
LIN {X 0,Y 195.923,Z 762.945,A -85,B 0,C 180,E1 -23899.783,E2 -23899.783} C_VEL
LIN {X 0,Y 186.021,Z 766.212,A -85,B 0,C 180,E1 -23902.808,E2 -23902.808} C_VEL
LIN {X 0,Y 177.061,Z 768.229,A -85,B 0,C 180,E1 -23906.241,E2 -23906.241} C_VEL
LIN {X 0,Y 169.195,Z 769.052,A -85,B 0,C 180,E1 -23910.102,E2 -23910.102} C_VEL
LIN {X 0,Y 162.383,Z 768.699,A -85,B 0,C 180,E1 -23914.354,E2 -23914.354} C_VEL
LIN {X 0,Y 159.36,Z 768.071,A -85,B 0,C 180,E1 -23916.615,E2 -23916.615} C_VEL
LIN {X 0,Y 154.703,Z 765.894,A -85,B 0,C 180,E1 -23921.458,E2 -23921.458} C_VEL
LIN {X 0,Y 151.337,Z 762.459,A -85,B 0,C 180,E1 -23926.573,E2 -23926.573} C_VEL
LIN {X 0,Y 149.342,Z 757.626,A -85,B 0,C 180,E1 -23931.884,E2 -23931.884} C_VEL
LIN {X 0,Y 148.823,Z 753.038,A -85,B 0,C 180,E1 -23935.938,E2 -23935.938} C_VEL
LIN {X 0,Y 148.718,Z 746.291,A -85,B 0,C 180,E1 -23940.677,E2 -23940.677} C_VEL
LIN {X 0,Y 148.877,Z 739.103,A -85,B 0,C 180,E1 -23944.739,E2 -23944.739} C_VEL
LIN {X 0,Y 149.327,Z 730.239,A -85,B 0,C 180,E1 -23948.781,E2 -23948.781} C_VEL
LIN {X 0,Y 150.188,Z 719.363,A -85,B 0,C 180,E1 -23952.843,E2 -23952.843} C_VEL
LIN {X 0,Y 151.118,Z 708.223,A -85,B 0,C 180,E1 -23956.203,E2 -23956.203} C_VEL
LIN {X 0,Y 152.534,Z 696.199,A -85,B 0,C 180,E1 -23959.165,E2 -23959.165} C_VEL
LIN {X 0,Y 153.971,Z 682.902,A -85,B 0,C 180,E1 -23961.769,E2 -23961.769} C_VEL
LIN {X 0,Y 155.319,Z 668.026,A -85,B 0,C 180,E1 -23964.031,E2 -23964.031} C_VEL
LIN {X 0,Y 156.603,Z 651.852,A -85,B 0,C 180,E1 -23965.815,E2 -23965.815} C_VEL
LIN {X 0,Y 161.296,Z 586.482,A -85,B 0,C 180,E1 -23971.433,E2 -23971.433} C_VEL
LIN {X 0,Y 158.793,Z 552.884,A -85,B 0,C 180,E1 -23974.479,E2 -23974.479} C_VEL
LIN {X 0,Y 154.638,Z 536.959,A -85,B 0,C 180,E1 -23976.215,E2 -23976.215} C_VEL
LIN {X 0,Y 152.303,Z 526.464,A -85,B 0,C 180,E1 -23981.742,E2 -23981.742} C_VEL
LIN {X 0,Y 150.2,Z 516.903,A -85,B 0,C 180,E1 -23987.164,E2 -23987.164} C_VEL
LIN {X 0,Y 150.18,Z 516.901,A -85,B 0,C 180,E1 -23992.707,E2 -23992.707} C_VEL
LIN {X 0,Y 150.221,Z 516.895,A -85,B 0,C 180,E1 -23997.364,E2 -23997.364} C_VEL
LIN {X 0,Y 150.247,Z 516.891,A -85,B 0,C 180,E1 -24002.717,E2 -24002.717} C_VEL
LIN {X 0,Y 150.352,Z 516.882,A -85,B 0,C 180,E1 -24009.207,E2 -24009.207} C_VEL
LIN {X 0,Y 150.384,Z 516.874,A -85,B 0,C 180,E1 -24013.716,E2 -24013.716} C_VEL
LIN {X 0,Y 150.691,Z 516.838,A -85,B 0,C 180,E1 -24019.248,E2 -24019.248} C_VEL
LIN {X 0,Y 150.765,Z 516.827,A -85,B 0,C 180,E1 -24021.961,E2 -24021.961} C_VEL
LIN {X 0,Y 151.221,Z 516.768,A -85,B 0,C 180,E1 -24030,E2 -24030} C_VEL
LIN {X 0,Y 150.764,Z 516.824,A -85,B 0,C 180,E1 -24038.039,E2 -24038.039} C_VEL
LIN {X 0,Y 150.636,Z 516.847,A -85,B 0,C 180,E1 -24041.546,E2 -24041.546} C_VEL
LIN {X 0,Y 150.392,Z 516.87,A -85,B 0,C 180,E1 -24046.283,E2 -24046.283} C_VEL
LIN {X 0,Y 150.353,Z 516.881,A -85,B 0,C 180,E1 -24050.794,E2 -24050.794} C_VEL
LIN {X 0,Y 150.245,Z 516.893,A -85,B 0,C 180,E1 -24057.282,E2 -24057.282} C_VEL
LIN {X 0,Y 150.218,Z 516.894,A -85,B 0,C 180,E1 -24062.634,E2 -24062.634} C_VEL
LIN {X 0,Y 150.212,Z 516.9,A -85,B 0,C 180,E1 -24067.462,E2 -24067.462} C_VEL
LIN {X 0,Y 150.155,Z 516.901,A -85,B 0,C 180,E1 -24071.507,E2 -24071.507} C_VEL
LIN {X 0,Y 150.246,Z 516.995,A -85,B 0,C 180,E1 -24076.975,E2 -24076.975} C_VEL
LIN {X 0,Y 153.836,Z 532.416,A -85,B 0,C 180,E1 -24082.529,E2 -24082.529} C_VEL
LIN {X 0,Y 157.046,Z 547.079,A -85,B 0,C 180,E1 -24087.519,E2 -24087.519} C_VEL
LIN {X 0,Y 157.088,Z 549.956,A -85,B 0,C 180,E1 -24088.44,E2 -24088.44} C_VEL
LIN {X 0,Y 156.651,Z 552.735,A -85,B 0,C 180,E1 -24089.304,E2 -24089.304} C_VEL
LIN {X 0,Y 157.822,Z 577.417,A -85,B 0,C 180,E1 -24091.432,E2 -24091.432} C_VEL
LIN {X 0,Y 158.735,Z 588.196,A -85,B 0,C 180,E1 -24092.363,E2 -24092.363} C_VEL
LIN {X 0,Y 154.827,Z 660.643,A -85,B 0,C 180,E1 -24098.62,E2 -24098.62} C_VEL
LIN {X 0,Y 153.943,Z 674.579,A -85,B 0,C 180,E1 -24100.151,E2 -24100.151} C_VEL
LIN {X 0,Y 152.864,Z 688.505,A -85,B 0,C 180,E1 -24102.267,E2 -24102.267} C_VEL
LIN {X 0,Y 151.753,Z 701.713,A -85,B 0,C 180,E1 -24104.9,E2 -24104.9} C_VEL
LIN {X 0,Y 150.83,Z 712.794,A -85,B 0,C 180,E1 -24107.657,E2 -24107.657} C_VEL
LIN {X 0,Y 149.964,Z 724.547,A -85,B 0,C 180,E1 -24111.294,E2 -24111.294} C_VEL
LIN {X 0,Y 149.463,Z 733.214,A -85,B 0,C 180,E1 -24114.604,E2 -24114.604} C_VEL
LIN {X 0,Y 149.186,Z 741.863,A -85,B 0,C 180,E1 -24118.65,E2 -24118.65} C_VEL
LIN {X 0,Y 149.052,Z 748.865,A -85,B 0,C 180,E1 -24122.703,E2 -24122.703} C_VEL
LIN {X 0,Y 149.169,Z 754.781,A -85,B 0,C 180,E1 -24127.028,E2 -24127.028} C_VEL
LIN {X 0,Y 150.36,Z 760.412,A -85,B 0,C 180,E1 -24132.142,E2 -24132.142} C_VEL
LIN {X 0,Y 152.114,Z 763.8,A -85,B 0,C 180,E1 -24136.094,E2 -24136.094} C_VEL
LIN {X 0,Y 155.861,Z 767.164,A -85,B 0,C 180,E1 -24141.145,E2 -24141.145} C_VEL
LIN {X 0,Y 160.869,Z 769.191,A -85,B 0,C 180,E1 -24145.905,E2 -24145.905} C_VEL
LIN {X 0,Y 167.449,Z 769.945,A -85,B 0,C 180,E1 -24150.242,E2 -24150.242} C_VEL
LIN {X 0,Y 175.201,Z 769.427,A -85,B 0,C 180,E1 -24154.166,E2 -24154.166} C_VEL
LIN {X 0,Y 184.028,Z 767.627,A -85,B 0,C 180,E1 -24157.665,E2 -24157.665} C_VEL
LIN {X 0,Y 193.746,Z 764.492,A -85,B 0,C 180,E1 -24160.764,E2 -24160.764} C_VEL
LIN {X 0,Y 204.26,Z 759.892,A -85,B 0,C 180,E1 -24163.483,E2 -24163.483} C_VEL
LIN {X 0,Y 205.255,Z 759.434,A -85,B 0,C 180,E1 -24164.024,E2 -24164.024} C_VEL
LIN {X 0,Y 194.407,Z 764.732,A -85,B 0,C 180,E1 -24166.617,E2 -24166.617} C_VEL
LIN {X 0,Y 184.459,Z 768.66,A -85,B 0,C 180,E1 -24169.631,E2 -24169.631} C_VEL
LIN {X 0,Y 175.497,Z 771.341,A -85,B 0,C 180,E1 -24173.08,E2 -24173.08} C_VEL
LIN {X 0,Y 167.549,Z 772.835,A -85,B 0,C 180,E1 -24176.955,E2 -24176.955} C_VEL
LIN {X 0,Y 160.989,Z 773.156,A -85,B 0,C 180,E1 -24181.301,E2 -24181.301} C_VEL
LIN {X 0,Y 155.773,Z 772.309,A -85,B 0,C 180,E1 -24186.043,E2 -24186.043} C_VEL
LIN {X 0,Y 152.014,Z 770.276,A -85,B 0,C 180,E1 -24191.118,E2 -24191.118} C_VEL
LIN {X 0,Y 149.965,Z 767.041,A -85,B 0,C 180,E1 -24196.448,E2 -24196.448} C_VEL
LIN {X 0,Y 149.389,Z 762.426,A -85,B 0,C 180,E1 -24201.887,E2 -24201.887} C_VEL
LIN {X 0,Y 149.586,Z 759.304,A -85,B 0,C 180,E1 -24204.774,E2 -24204.774} C_VEL
LIN {X 0,Y 149.363,Z 758.003,A -85,B 0,C 180,E1 -24206.153,E2 -24206.153} C_VEL
LIN {X 0,Y 148.581,Z 757.303,A -85,B 0,C 180,E1 -24207.58,E2 -24207.58} C_VEL
LIN {X 0,Y 146.821,Z 757.172,A -85,B 0,C 180,E1 -24209.756,E2 -24209.756} C_VEL
LIN {X 0,Y 144.81,Z 757.951,A -85,B 0,C 180,E1 -24211.985,E2 -24211.985} C_VEL
LIN {X 0,Y 142.693,Z 759.962,A -85,B 0,C 180,E1 -24215.04,E2 -24215.04} C_VEL
LIN {X 0,Y 142.263,Z 761.261,A -85,B 0,C 180,E1 -24216.591,E2 -24216.591} C_VEL
LIN {X 0,Y 142.323,Z 765.1,A -85,B 0,C 180,E1 -24221.392,E2 -24221.392} C_VEL
LIN {X 0,Y 143.744,Z 768.568,A -85,B 0,C 180,E1 -24227.059,E2 -24227.059} C_VEL
LIN {X 0,Y 146.809,Z 770.944,A -85,B 0,C 180,E1 -24232.518,E2 -24232.518} C_VEL
LIN {X 0,Y 151.414,Z 772.285,A -85,B 0,C 180,E1 -24237.656,E2 -24237.656} C_VEL
LIN {X 0,Y 157.4,Z 772.655,A -85,B 0,C 180,E1 -24242.399,E2 -24242.399} C_VEL
LIN {X 0,Y 164.581,Z 772.06,A -85,B 0,C 180,E1 -24246.715,E2 -24246.715} C_VEL
LIN {X 0,Y 173.059,Z 770.507,A -85,B 0,C 180,E1 -24250.524,E2 -24250.524} C_VEL
LIN {X 0,Y 182.584,Z 767.919,A -85,B 0,C 180,E1 -24253.857,E2 -24253.857} C_VEL
LIN {X 0,Y 192.938,Z 764.268,A -85,B 0,C 180,E1 -24256.763,E2 -24256.763} C_VEL
LIN {X 0,Y 193.923,Z 763.831,A -85,B 0,C 180,E1 -24257.605,E2 -24257.605} C_VEL
LIN {X 0,Y 185.472,Z 766.375,A -85,B 0,C 180,E1 -24259.896,E2 -24259.896} C_VEL
LIN {X 0,Y 174.969,Z 768.61,A -85,B 0,C 180,E1 -24263.451,E2 -24263.451} C_VEL
LIN {X 0,Y 167.003,Z 769.401,A -85,B 0,C 180,E1 -24266.833,E2 -24266.833} C_VEL
LIN {X 0,Y 159.405,Z 769.176,A -85,B 0,C 180,E1 -24270.989,E2 -24270.989} C_VEL
LIN {X 0,Y 152.889,Z 767.774,A -85,B 0,C 180,E1 -24275.562,E2 -24275.562} C_VEL
LIN {X 0,Y 148.026,Z 765.201,A -85,B 0,C 180,E1 -24280.589,E2 -24280.589} C_VEL
LIN {X 0,Y 144.533,Z 761.385,A -85,B 0,C 180,E1 -24285.929,E2 -24285.929} C_VEL
LIN {X 0,Y 142.475,Z 756.174,A -85,B 0,C 180,E1 -24291.49,E2 -24291.49} C_VEL
LIN {X 0,Y 141.953,Z 751.277,A -85,B 0,C 180,E1 -24295.741,E2 -24295.741} C_VEL
LIN {X 0,Y 141.853,Z 745.245,A -85,B 0,C 180,E1 -24300,E2 -24300} C_VEL
LIN {X 0,Y 142.004,Z 737.877,A -85,B 0,C 180,E1 -24304.257,E2 -24304.257} C_VEL
LIN {X 0,Y 142.39,Z 728.883,A -85,B 0,C 180,E1 -24308.515,E2 -24308.515} C_VEL
LIN {X 0,Y 143.188,Z 718.727,A -85,B 0,C 180,E1 -24312.4,E2 -24312.4} C_VEL
LIN {X 0,Y 144.106,Z 707.455,A -85,B 0,C 180,E1 -24315.922,E2 -24315.922} C_VEL
LIN {X 0,Y 145.484,Z 695.389,A -85,B 0,C 180,E1 -24319.031,E2 -24319.031} C_VEL
LIN {X 0,Y 146.941,Z 682.097,A -85,B 0,C 180,E1 -24321.757,E2 -24321.757} C_VEL
LIN {X 0,Y 148.173,Z 668.315,A -85,B 0,C 180,E1 -24323.962,E2 -24323.962} C_VEL
LIN {X 0,Y 149.453,Z 652.535,A -85,B 0,C 180,E1 -24325.804,E2 -24325.804} C_VEL
LIN {X 0,Y 154.221,Z 586.399,A -85,B 0,C 180,E1 -24331.785,E2 -24331.785} C_VEL
LIN {X 0,Y 151.816,Z 553.975,A -85,B 0,C 180,E1 -24334.879,E2 -24334.879} C_VEL
LIN {X 0,Y 147.319,Z 536.752,A -85,B 0,C 180,E1 -24336.914,E2 -24336.914} C_VEL
LIN {X 0,Y 145.17,Z 527.015,A -85,B 0,C 180,E1 -24342.286,E2 -24342.286} C_VEL
LIN {X 0,Y 143.149,Z 517.782,A -85,B 0,C 180,E1 -24347.777,E2 -24347.777} C_VEL
LIN {X 0,Y 143.089,Z 517.783,A -85,B 0,C 180,E1 -24353.885,E2 -24353.885} C_VEL
LIN {X 0,Y 143.188,Z 517.77,A -85,B 0,C 180,E1 -24357.322,E2 -24357.322} C_VEL
LIN {X 0,Y 143.194,Z 517.77,A -85,B 0,C 180,E1 -24362.061,E2 -24362.061} C_VEL
LIN {X 0,Y 143.278,Z 517.762,A -85,B 0,C 180,E1 -24368.745,E2 -24368.745} C_VEL
LIN {X 0,Y 143.318,Z 517.751,A -85,B 0,C 180,E1 -24372.889,E2 -24372.889} C_VEL
LIN {X 0,Y 143.604,Z 517.72,A -85,B 0,C 180,E1 -24378.711,E2 -24378.711} C_VEL
LIN {X 0,Y 143.686,Z 517.707,A -85,B 0,C 180,E1 -24381.562,E2 -24381.562} C_VEL
LIN {X 0,Y 144.18,Z 517.645,A -85,B 0,C 180,E1 -24390,E2 -24390} C_VEL
LIN {X 0,Y 143.686,Z 517.705,A -85,B 0,C 180,E1 -24398.438,E2 -24398.438} C_VEL
LIN {X 0,Y 143.572,Z 517.726,A -85,B 0,C 180,E1 -24401.757,E2 -24401.757} C_VEL
LIN {X 0,Y 143.324,Z 517.751,A -85,B 0,C 180,E1 -24407.11,E2 -24407.11} C_VEL
LIN {X 0,Y 143.279,Z 517.764,A -85,B 0,C 180,E1 -24411.256,E2 -24411.256} C_VEL
LIN {X 0,Y 143.191,Z 517.773,A -85,B 0,C 180,E1 -24417.937,E2 -24417.937} C_VEL
LIN {X 0,Y 143.169,Z 517.771,A -85,B 0,C 180,E1 -24423.435,E2 -24423.435} C_VEL
LIN {X 0,Y 143.076,Z 517.786,A -85,B 0,C 180,E1 -24429.685,E2 -24429.685} C_VEL
LIN {X 0,Y 143.152,Z 517.777,A -85,B 0,C 180,E1 -24436.352,E2 -24436.352} C_VEL
LIN {X 0,Y 146.517,Z 532.196,A -85,B 0,C 180,E1 -24441.815,E2 -24441.815} C_VEL
LIN {X 0,Y 149.64,Z 546.435,A -85,B 0,C 180,E1 -24446.86,E2 -24446.86} C_VEL
LIN {X 0,Y 150.168,Z 549.425,A -85,B 0,C 180,E1 -24447.88,E2 -24447.88} C_VEL
LIN {X 0,Y 149.62,Z 552.974,A -85,B 0,C 180,E1 -24448.997,E2 -24448.997} C_VEL
LIN {X 0,Y 150.761,Z 577.752,A -85,B 0,C 180,E1 -24451.242,E2 -24451.242} C_VEL
LIN {X 0,Y 151.645,Z 588.596,A -85,B 0,C 180,E1 -24452.223,E2 -24452.223} C_VEL
LIN {X 0,Y 147.845,Z 657.736,A -85,B 0,C 180,E1 -24458.566,E2 -24458.566} C_VEL
LIN {X 0,Y 146.98,Z 673.016,A -85,B 0,C 180,E1 -24460.263,E2 -24460.263} C_VEL
LIN {X 0,Y 145.899,Z 687.275,A -85,B 0,C 180,E1 -24462.478,E2 -24462.478} C_VEL
LIN {X 0,Y 144.775,Z 700.77,A -85,B 0,C 180,E1 -24465.235,E2 -24465.235} C_VEL
LIN {X 0,Y 143.894,Z 711.595,A -85,B 0,C 180,E1 -24468.019,E2 -24468.019} C_VEL
LIN {X 0,Y 143.114,Z 722.593,A -85,B 0,C 180,E1 -24471.528,E2 -24471.528} C_VEL
LIN {X 0,Y 142.646,Z 731.675,A -85,B 0,C 180,E1 -24475.054,E2 -24475.054} C_VEL
LIN {X 0,Y 142.358,Z 740.621,A -85,B 0,C 180,E1 -24479.293,E2 -24479.293} C_VEL
LIN {X 0,Y 142.262,Z 747.732,A -85,B 0,C 180,E1 -24483.54,E2 -24483.54} C_VEL
LIN {X 0,Y 142.474,Z 754.344,A -85,B 0,C 180,E1 -24488.51,E2 -24488.51} C_VEL
LIN {X 0,Y 144.154,Z 760.305,A -85,B 0,C 180,E1 -24494.109,E2 -24494.109} C_VEL
LIN {X 0,Y 147.169,Z 764.739,A -85,B 0,C 180,E1 -24499.529,E2 -24499.529} C_VEL
LIN {X 0,Y 151.675,Z 767.821,A -85,B 0,C 180,E1 -24504.647,E2 -24504.647} C_VEL
LIN {X 0,Y 157.787,Z 769.675,A -85,B 0,C 180,E1 -24509.337,E2 -24509.337} C_VEL
LIN {X 0,Y 165.213,Z 770.289,A -85,B 0,C 180,E1 -24513.574,E2 -24513.574} C_VEL
LIN {X 0,Y 173.828,Z 769.658,A -85,B 0,C 180,E1 -24517.334,E2 -24517.334} C_VEL
LIN {X 0,Y 183.445,Z 767.755,A -85,B 0,C 180,E1 -24520.639,E2 -24520.639} C_VEL
LIN {X 0,Y 194.858,Z 764.142,A -85,B 0,C 180,E1 -24523.834,E2 -24523.834} C_VEL
LIN {X 0,Y 184.177,Z 768.099,A -85,B 0,C 180,E1 -24526.618,E2 -24526.618} C_VEL
LIN {X 0,Y 174.415,Z 770.824,A -85,B 0,C 180,E1 -24529.856,E2 -24529.856} C_VEL
LIN {X 0,Y 165.666,Z 772.392,A -85,B 0,C 180,E1 -24533.564,E2 -24533.564} C_VEL
LIN {X 0,Y 158.044,Z 772.823,A -85,B 0,C 180,E1 -24537.749,E2 -24537.749} C_VEL
LIN {X 0,Y 151.88,Z 772.129,A -85,B 0,C 180,E1 -24542.436,E2 -24542.436} C_VEL
LIN {X 0,Y 147.193,Z 770.298,A -85,B 0,C 180,E1 -24547.544,E2 -24547.544} C_VEL
LIN {X 0,Y 144.121,Z 767.28,A -85,B 0,C 180,E1 -24552.987,E2 -24552.987} C_VEL
LIN {X 0,Y 142.779,Z 763.005,A -85,B 0,C 180,E1 -24558.645,E2 -24558.645} C_VEL
LIN {X 0,Y 142.88,Z 757.21,A -85,B 0,C 180,E1 -24564.354,E2 -24564.354} C_VEL
LIN {X 0,Y 143.504,Z 751.972,A -85,B 0,C 180,E1 -24568.422,E2 -24568.422} C_VEL
LIN {X 0,Y 142.473,Z 759.004,A -85,B 0,C 180,E1 -24574.244,E2 -24574.244} C_VEL
LIN {X 0,Y 142.263,Z 761.261,A -85,B 0,C 180,E1 -24576.591,E2 -24576.591} C_VEL
LIN {X 0,Y 141.522,Z 762.987,A -85,B 0,C 180,E1 -24578.856,E2 -24578.856} C_VEL
LIN {X 0,Y 139.065,Z 764.961,A -85,B 0,C 180,E1 -24582.704,E2 -24582.704} C_VEL
LIN {X 0,Y 137.481,Z 766.225,A -85,B 0,C 180,E1 -24585.901,E2 -24585.901} C_VEL
LIN {X 0,Y 137.38,Z 767.28,A -85,B 0,C 180,E1 -24588.337,E2 -24588.337} C_VEL
LIN {X 0,Y 137.664,Z 767.659,A -85,B 0,C 180,E1 -24589.136,E2 -24589.136} C_VEL
LIN {X 0,Y 140.343,Z 769.751,A -85,B 0,C 180,E1 -24593.617,E2 -24593.617} C_VEL
LIN {X 0,Y 145.172,Z 771.478,A -85,B 0,C 180,E1 -24598.955,E2 -24598.955} C_VEL
LIN {X 0,Y 151.47,Z 772.205,A -85,B 0,C 180,E1 -24603.834,E2 -24603.834} C_VEL
LIN {X 0,Y 158.953,Z 772.003,A -85,B 0,C 180,E1 -24608.244,E2 -24608.244} C_VEL
LIN {X 0,Y 167.744,Z 770.875,A -85,B 0,C 180,E1 -24612.095,E2 -24612.095} C_VEL
LIN {X 0,Y 177.584,Z 768.797,A -85,B 0,C 180,E1 -24615.428,E2 -24615.428} C_VEL
LIN {X 0,Y 182.79,Z 767.365,A -85,B 0,C 180,E1 -24616.931,E2 -24616.931} C_VEL
LIN {X 0,Y 183.208,Z 767.183,A -85,B 0,C 180,E1 -24617.621,E2 -24617.621} C_VEL
LIN {X 0,Y 175.071,Z 768.751,A -85,B 0,C 180,E1 -24620.036,E2 -24620.036} C_VEL
LIN {X 0,Y 165.516,Z 769.764,A -85,B 0,C 180,E1 -24623.526,E2 -24623.526} C_VEL
LIN {X 0,Y 157.064,Z 769.644,A -85,B 0,C 180,E1 -24627.523,E2 -24627.523} C_VEL
LIN {X 0,Y 149.723,Z 768.393,A -85,B 0,C 180,E1 -24632.005,E2 -24632.005} C_VEL
LIN {X 0,Y 143.749,Z 765.98,A -85,B 0,C 180,E1 -24636.975,E2 -24636.975} C_VEL
LIN {X 0,Y 139.435,Z 762.407,A -85,B 0,C 180,E1 -24642.397,E2 -24642.397} C_VEL
LIN {X 0,Y 136.503,Z 757.504,A -85,B 0,C 180,E1 -24648.115,E2 -24648.115} C_VEL
LIN {X 0,Y 135.256,Z 751.164,A -85,B 0,C 180,E1 -24654.035,E2 -24654.035} C_VEL
LIN {X 0,Y 135.026,Z 744.156,A -85,B 0,C 180,E1 -24659.254,E2 -24659.254} C_VEL
LIN {X 0,Y 135.149,Z 736.591,A -85,B 0,C 180,E1 -24663.727,E2 -24663.727} C_VEL
LIN {X 0,Y 135.551,Z 727.06,A -85,B 0,C 180,E1 -24668.297,E2 -24668.297} C_VEL
LIN {X 0,Y 136.364,Z 715.95,A -85,B 0,C 180,E1 -24672.652,E2 -24672.652} C_VEL
LIN {X 0,Y 137.338,Z 704.124,A -85,B 0,C 180,E1 -24676.347,E2 -24676.347} C_VEL
LIN {X 0,Y 138.803,Z 691.277,A -85,B 0,C 180,E1 -24679.599,E2 -24679.599} C_VEL
LIN {X 0,Y 140.221,Z 677.955,A -85,B 0,C 180,E1 -24682.274,E2 -24682.274} C_VEL
LIN {X 0,Y 141.526,Z 663.069,A -85,B 0,C 180,E1 -24684.575,E2 -24684.575} C_VEL
LIN {X 0,Y 142.941,Z 644.792,A -85,B 0,C 180,E1 -24686.6,E2 -24686.6} C_VEL
LIN {X 0,Y 147.203,Z 586.947,A -85,B 0,C 180,E1 -24692.106,E2 -24692.106} C_VEL
LIN {X 0,Y 144.957,Z 555.667,A -85,B 0,C 180,E1 -24695.25,E2 -24695.25} C_VEL
LIN {X 0,Y 140.073,Z 536.704,A -85,B 0,C 180,E1 -24697.548,E2 -24697.548} C_VEL
LIN {X 0,Y 137.767,Z 526.391,A -85,B 0,C 180,E1 -24703.55,E2 -24703.55} C_VEL
LIN {X 0,Y 136.077,Z 518.661,A -85,B 0,C 180,E1 -24708.446,E2 -24708.446} C_VEL
LIN {X 0,Y 136.028,Z 518.666,A -85,B 0,C 180,E1 -24711.684,E2 -24711.684} C_VEL
LIN {X 0,Y 136.058,Z 518.656,A -85,B 0,C 180,E1 -24715.738,E2 -24715.738} C_VEL
LIN {X 0,Y 136.149,Z 518.647,A -85,B 0,C 180,E1 -24722.317,E2 -24722.317} C_VEL
LIN {X 0,Y 136.245,Z 518.638,A -85,B 0,C 180,E1 -24728.833,E2 -24728.833} C_VEL
LIN {X 0,Y 136.287,Z 518.631,A -85,B 0,C 180,E1 -24735.058,E2 -24735.058} C_VEL
LIN {X 0,Y 136.503,Z 518.605,A -85,B 0,C 180,E1 -24738.115,E2 -24738.115} C_VEL
LIN {X 0,Y 136.61,Z 518.587,A -85,B 0,C 180,E1 -24741.121,E2 -24741.121} C_VEL
LIN {X 0,Y 137.137,Z 518.522,A -85,B 0,C 180,E1 -24750,E2 -24750} C_VEL
LIN {X 0,Y 136.61,Z 518.587,A -85,B 0,C 180,E1 -24758.878,E2 -24758.878} C_VEL
LIN {X 0,Y 136.494,Z 518.607,A -85,B 0,C 180,E1 -24761.959,E2 -24761.959} C_VEL
LIN {X 0,Y 136.258,Z 518.634,A -85,B 0,C 180,E1 -24768.027,E2 -24768.027} C_VEL
LIN {X 0,Y 136.2,Z 518.644,A -85,B 0,C 180,E1 -24771.75,E2 -24771.75} C_VEL
LIN {X 0,Y 136.101,Z 518.656,A -85,B 0,C 180,E1 -24778.616,E2 -24778.616} C_VEL
LIN {X 0,Y 136.079,Z 518.654,A -85,B 0,C 180,E1 -24784.619,E2 -24784.619} C_VEL
LIN {X 0,Y 136.051,Z 518.663,A -85,B 0,C 180,E1 -24789.208,E2 -24789.208} C_VEL
LIN {X 0,Y 136.112,Z 518.726,A -85,B 0,C 180,E1 -24795.921,E2 -24795.921} C_VEL
LIN {X 0,Y 139.721,Z 534.301,A -85,B 0,C 180,E1 -24801.951,E2 -24801.951} C_VEL
LIN {X 0,Y 142.895,Z 548.766,A -85,B 0,C 180,E1 -24807.247,E2 -24807.247} C_VEL
LIN {X 0,Y 142.843,Z 551.186,A -85,B 0,C 180,E1 -24808.068,E2 -24808.068} C_VEL
LIN {X 0,Y 142.563,Z 553.276,A -85,B 0,C 180,E1 -24808.724,E2 -24808.724} C_VEL
LIN {X 0,Y 143.538,Z 575.746,A -85,B 0,C 180,E1 -24810.849,E2 -24810.849} C_VEL
LIN {X 0,Y 144.532,Z 589.04,A -85,B 0,C 180,E1 -24812.119,E2 -24812.119} C_VEL
LIN {X 0,Y 140.651,Z 660.836,A -85,B 0,C 180,E1 -24819.144,E2 -24819.144} C_VEL
LIN {X 0,Y 139.738,Z 675.131,A -85,B 0,C 180,E1 -24820.919,E2 -24820.919} C_VEL
LIN {X 0,Y 138.76,Z 687.818,A -85,B 0,C 180,E1 -24823.068,E2 -24823.068} C_VEL
LIN {X 0,Y 137.801,Z 699.962,A -85,B 0,C 180,E1 -24825.701,E2 -24825.701} C_VEL
LIN {X 0,Y 136.871,Z 712.049,A -85,B 0,C 180,E1 -24828.988,E2 -24828.988} C_VEL
LIN {X 0,Y 136.183,Z 722.728,A -85,B 0,C 180,E1 -24832.587,E2 -24832.587} C_VEL
LIN {X 0,Y 135.811,Z 731.698,A -85,B 0,C 180,E1 -24836.291,E2 -24836.291} C_VEL
LIN {X 0,Y 135.584,Z 740.488,A -85,B 0,C 180,E1 -24840.743,E2 -24840.743} C_VEL
LIN {X 0,Y 135.526,Z 746.481,A -85,B 0,C 180,E1 -24844.461,E2 -24844.461} C_VEL
LIN {X 0,Y 135.9,Z 753.422,A -85,B 0,C 180,E1 -24849.798,E2 -24849.798} C_VEL
LIN {X 0,Y 137.449,Z 758.78,A -85,B 0,C 180,E1 -24854.813,E2 -24854.813} C_VEL
LIN {X 0,Y 140.586,Z 763.622,A -85,B 0,C 180,E1 -24860.483,E2 -24860.483} C_VEL
LIN {X 0,Y 145.308,Z 767.127,A -85,B 0,C 180,E1 -24865.804,E2 -24865.804} C_VEL
LIN {X 0,Y 151.657,Z 769.433,A -85,B 0,C 180,E1 -24870.648,E2 -24870.648} C_VEL
LIN {X 0,Y 159.358,Z 770.539,A -85,B 0,C 180,E1 -24874.983,E2 -24874.983} C_VEL
LIN {X 0,Y 168.283,Z 770.427,A -85,B 0,C 180,E1 -24878.788,E2 -24878.788} C_VEL
LIN {X 0,Y 178.191,Z 769.057,A -85,B 0,C 180,E1 -24882.105,E2 -24882.105} C_VEL
LIN {X 0,Y 183.462,Z 767.906,A -85,B 0,C 180,E1 -24883.594,E2 -24883.594} C_VEL
LIN {X 0,Y 179.12,Z 769.126,A -85,B 0,C 180,E1 -24885.069,E2 -24885.069} C_VEL
LIN {X 0,Y 169.069,Z 771.297,A -85,B 0,C 180,E1 -24888.31,E2 -24888.31} C_VEL
LIN {X 0,Y 160.018,Z 772.35,A -85,B 0,C 180,E1 -24892.057,E2 -24892.057} C_VEL
LIN {X 0,Y 152.113,Z 772.298,A -85,B 0,C 180,E1 -24896.328,E2 -24896.328} C_VEL
LIN {X 0,Y 145.681,Z 771.173,A -85,B 0,C 180,E1 -24901.156,E2 -24901.156} C_VEL
LIN {X 0,Y 140.778,Z 768.957,A -85,B 0,C 180,E1 -24906.461,E2 -24906.461} C_VEL
LIN {X 0,Y 137.541,Z 765.571,A -85,B 0,C 180,E1 -24912.146,E2 -24912.146} C_VEL
LIN {X 0,Y 136.13,Z 760.898,A -85,B 0,C 180,E1 -24918.082,E2 -24918.082} C_VEL
LIN {X 0,Y 136.139,Z 756.461,A -85,B 0,C 180,E1 -24922.585,E2 -24922.585} C_VEL
LIN {X 0,Y 136.847,Z 749.857,A -85,B 0,C 180,E1 -24927.793,E2 -24927.793} C_VEL
LIN {X 0,Y 136.963,Z 749.276,A -85,B 0,C 180,E1 -24928.254,E2 -24928.254} C_VEL
LIN {X 0,Y 135.907,Z 755.151,A -85,B 0,C 180,E1 -24932.964,E2 -24932.964} C_VEL
LIN {X 0,Y 135.464,Z 760.127,A -85,B 0,C 180,E1 -24938.001,E2 -24938.001} C_VEL
LIN {X 0,Y 135.861,Z 764.35,A -85,B 0,C 180,E1 -24943.461,E2 -24943.461} C_VEL
LIN {X 0,Y 137.664,Z 767.659,A -85,B 0,C 180,E1 -24949.136,E2 -24949.136} C_VEL
LIN {X 0,Y 138.301,Z 768.699,A -85,B 0,C 180,E1 -24951.538,E2 -24951.538} C_VEL
LIN {X 0,Y 138.277,Z 769.7,A -85,B 0,C 180,E1 -24955.626,E2 -24955.626} C_VEL
LIN {X 0,Y 138.722,Z 770.266,A -85,B 0,C 180,E1 -24958.9,E2 -24958.9} C_VEL
LIN {X 0,Y 140.13,Z 770.702,A -85,B 0,C 180,E1 -24961.253,E2 -24961.253} C_VEL
LIN {X 0,Y 140.899,Z 770.882,A -85,B 0,C 180,E1 -24961.989,E2 -24961.989} C_VEL
LIN {X 0,Y 149.401,Z 771.794,A -85,B 0,C 180,E1 -24967.701,E2 -24967.701} C_VEL
LIN {X 0,Y 157.876,Z 771.538,A -85,B 0,C 180,E1 -24971.893,E2 -24971.893} C_VEL
LIN {X 0,Y 167.518,Z 770.39,A -85,B 0,C 180,E1 -24975.497,E2 -24975.497} C_VEL
LIN {X 0,Y 172.706,Z 769.455,A -85,B 0,C 180,E1 -24977.096,E2 -24977.096} C_VEL
LIN {X 0,Y 169.72,Z 769.745,A -85,B 0,C 180,E1 -24978.505,E2 -24978.505} C_VEL
LIN {X 0,Y 159.88,Z 770.257,A -85,B 0,C 180,E1 -24982.018,E2 -24982.018} C_VEL
LIN {X 0,Y 151.133,Z 769.676,A -85,B 0,C 180,E1 -24986.081,E2 -24986.081} C_VEL
LIN {X 0,Y 143.513,Z 767.982,A -85,B 0,C 180,E1 -24990.678,E2 -24990.678} C_VEL
LIN {X 0,Y 137.289,Z 765.166,A -85,B 0,C 180,E1 -24995.825,E2 -24995.825} C_VEL
LIN {X 0,Y 132.795,Z 761.189,A -85,B 0,C 180,E1 -25001.486,E2 -25001.486} C_VEL
LIN {X 0,Y 129.764,Z 755.864,A -85,B 0,C 180,E1 -25007.488,E2 -25007.488} C_VEL
LIN {X 0,Y 128.468,Z 749.139,A -85,B 0,C 180,E1 -25013.718,E2 -25013.718} C_VEL
LIN {X 0,Y 128.262,Z 742.82,A -85,B 0,C 180,E1 -25018.43,E2 -25018.43} C_VEL
LIN {X 0,Y 128.343,Z 735.155,A -85,B 0,C 180,E1 -25023.139,E2 -25023.139} C_VEL
LIN {X 0,Y 128.678,Z 725.999,A -85,B 0,C 180,E1 -25027.681,E2 -25027.681} C_VEL
LIN {X 0,Y 129.44,Z 714.773,A -85,B 0,C 180,E1 -25032.223,E2 -25032.223} C_VEL
LIN {X 0,Y 130.353,Z 703.088,A -85,B 0,C 180,E1 -25036.04,E2 -25036.04} C_VEL
LIN {X 0,Y 131.805,Z 690.271,A -85,B 0,C 180,E1 -25039.467,E2 -25039.467} C_VEL
LIN {X 0,Y 133.236,Z 676.637,A -85,B 0,C 180,E1 -25042.28,E2 -25042.28} C_VEL
LIN {X 0,Y 134.555,Z 661.305,A -85,B 0,C 180,E1 -25044.699,E2 -25044.699} C_VEL
LIN {X 0,Y 136.256,Z 638.622,A -85,B 0,C 180,E1 -25047.243,E2 -25047.243} C_VEL
LIN {X 0,Y 140.128,Z 586.979,A -85,B 0,C 180,E1 -25052.48,E2 -25052.48} C_VEL
LIN {X 0,Y 137.9,Z 556.56,A -85,B 0,C 180,E1 -25055.692,E2 -25055.692} C_VEL
LIN {X 0,Y 132.802,Z 536.689,A -85,B 0,C 180,E1 -25058.191,E2 -25058.191} C_VEL
LIN {X 0,Y 130.515,Z 526.536,A -85,B 0,C 180,E1 -25064.429,E2 -25064.429} C_VEL
LIN {X 0,Y 129.019,Z 519.541,A -85,B 0,C 180,E1 -25069.051,E2 -25069.051} C_VEL
LIN {X 0,Y 128.961,Z 519.542,A -85,B 0,C 180,E1 -25074.831,E2 -25074.831} C_VEL
LIN {X 0,Y 129.052,Z 519.534,A -85,B 0,C 180,E1 -25080.651,E2 -25080.651} C_VEL
LIN {X 0,Y 129.109,Z 519.528,A -85,B 0,C 180,E1 -25087.727,E2 -25087.727} C_VEL
LIN {X 0,Y 129.162,Z 519.519,A -85,B 0,C 180,E1 -25090.945,E2 -25090.945} C_VEL
LIN {X 0,Y 129.42,Z 519.488,A -85,B 0,C 180,E1 -25097.815,E2 -25097.815} C_VEL
LIN {X 0,Y 129.532,Z 519.469,A -85,B 0,C 180,E1 -25100.632,E2 -25100.632} C_VEL
LIN {X 0,Y 130.093,Z 519.399,A -85,B 0,C 180,E1 -25110,E2 -25110} C_VEL
LIN {X 0,Y 129.532,Z 519.47,A -85,B 0,C 180,E1 -25119.368,E2 -25119.368} C_VEL
LIN {X 0,Y 129.396,Z 519.491,A -85,B 0,C 180,E1 -25122.548,E2 -25122.548} C_VEL
LIN {X 0,Y 129.164,Z 519.518,A -85,B 0,C 180,E1 -25129.054,E2 -25129.054} C_VEL
LIN {X 0,Y 129.109,Z 519.526,A -85,B 0,C 180,E1 -25132.398,E2 -25132.398} C_VEL
LIN {X 0,Y 129.036,Z 519.538,A -85,B 0,C 180,E1 -25139.373,E2 -25139.373} C_VEL
LIN {X 0,Y 128.993,Z 519.538,A -85,B 0,C 180,E1 -25145.189,E2 -25145.189} C_VEL
LIN {X 0,Y 128.951,Z 519.544,A -85,B 0,C 180,E1 -25150.845,E2 -25150.845} C_VEL
LIN {X 0,Y 129.044,Z 519.575,A -85,B 0,C 180,E1 -25155.35,E2 -25155.35} C_VEL
LIN {X 0,Y 132.657,Z 535.241,A -85,B 0,C 180,E1 -25161.686,E2 -25161.686} C_VEL
LIN {X 0,Y 135.825,Z 549.59,A -85,B 0,C 180,E1 -25167.119,E2 -25167.119} C_VEL
LIN {X 0,Y 135.494,Z 553.534,A -85,B 0,C 180,E1 -25168.434,E2 -25168.434} C_VEL
LIN {X 0,Y 136.693,Z 579.4,A -85,B 0,C 180,E1 -25171.046,E2 -25171.046} C_VEL
LIN {X 0,Y 137.422,Z 589.446,A -85,B 0,C 180,E1 -25172.056,E2 -25172.056} C_VEL
LIN {X 0,Y 133.821,Z 655.642,A -85,B 0,C 180,E1 -25178.935,E2 -25178.935} C_VEL
LIN {X 0,Y 132.956,Z 671.814,A -85,B 0,C 180,E1 -25180.909,E2 -25180.909} C_VEL
LIN {X 0,Y 131.988,Z 685.057,A -85,B 0,C 180,E1 -25183.13,E2 -25183.13} C_VEL
LIN {X 0,Y 130.967,Z 697.885,A -85,B 0,C 180,E1 -25185.935,E2 -25185.935} C_VEL
LIN {X 0,Y 130.127,Z 709.425,A -85,B 0,C 180,E1 -25189.104,E2 -25189.104} C_VEL
LIN {X 0,Y 129.425,Z 720.652,A -85,B 0,C 180,E1 -25192.982,E2 -25192.982} C_VEL
LIN {X 0,Y 129.074,Z 729.94,A -85,B 0,C 180,E1 -25196.879,E2 -25196.879} C_VEL
LIN {X 0,Y 128.912,Z 737.627,A -85,B 0,C 180,E1 -25200.781,E2 -25200.781} C_VEL
LIN {X 0,Y 128.856,Z 745.063,A -85,B 0,C 180,E1 -25205.477,E2 -25205.477} C_VEL
LIN {X 0,Y 129.525,Z 752.778,A -85,B 0,C 180,E1 -25211.582,E2 -25211.582} C_VEL
LIN {X 0,Y 131.421,Z 758.462,A -85,B 0,C 180,E1 -25217.105,E2 -25217.105} C_VEL
LIN {X 0,Y 135.21,Z 763.416,A -85,B 0,C 180,E1 -25222.945,E2 -25222.945} C_VEL
LIN {X 0,Y 139.005,Z 766.229,A -85,B 0,C 180,E1 -25227.067,E2 -25227.067} C_VEL
LIN {X 0,Y 145.616,Z 769,A -85,B 0,C 180,E1 -25232.067,E2 -25232.067} C_VEL
LIN {X 0,Y 153.609,Z 770.583,A -85,B 0,C 180,E1 -25236.497,E2 -25236.497} C_VEL
LIN {X 0,Y 162.828,Z 770.984,A -85,B 0,C 180,E1 -25240.348,E2 -25240.348} C_VEL
LIN {X 0,Y 173.038,Z 770.167,A -85,B 0,C 180,E1 -25243.667,E2 -25243.667} C_VEL
LIN {X 0,Y 163.843,Z 771.551,A -85,B 0,C 180,E1 -25246.661,E2 -25246.661} C_VEL
LIN {X 0,Y 154.495,Z 772.095,A -85,B 0,C 180,E1 -25250.442,E2 -25250.442} C_VEL
LIN {X 0,Y 146.28,Z 771.576,A -85,B 0,C 180,E1 -25254.792,E2 -25254.792} C_VEL
LIN {X 0,Y 139.594,Z 770.022,A -85,B 0,C 180,E1 -25259.771,E2 -25259.771} C_VEL
LIN {X 0,Y 134.448,Z 767.389,A -85,B 0,C 180,E1 -25265.28,E2 -25265.28} C_VEL
LIN {X 0,Y 131.048,Z 763.616,A -85,B 0,C 180,E1 -25271.23,E2 -25271.23} C_VEL
LIN {X 0,Y 129.566,Z 758.575,A -85,B 0,C 180,E1 -25277.519,E2 -25277.519} C_VEL
LIN {X 0,Y 129.721,Z 752.061,A -85,B 0,C 180,E1 -25283.78,E2 -25283.78} C_VEL
LIN {X 0,Y 130.475,Z 746.427,A -85,B 0,C 180,E1 -25288.071,E2 -25288.071} C_VEL
LIN {X 0,Y 129.117,Z 754.36,A -85,B 0,C 180,E1 -25294.683,E2 -25294.683} C_VEL
LIN {X 0,Y 128.773,Z 759.873,A -85,B 0,C 180,E1 -25300.771,E2 -25300.771} C_VEL
LIN {X 0,Y 129.586,Z 763.456,A -85,B 0,C 180,E1 -25305.734,E2 -25305.734} C_VEL
LIN {X 0,Y 132.068,Z 766.988,A -85,B 0,C 180,E1 -25311.871,E2 -25311.871} C_VEL
LIN {X 0,Y 136.326,Z 769.546,A -85,B 0,C 180,E1 -25317.644,E2 -25317.644} C_VEL
LIN {X 0,Y 140.899,Z 770.882,A -85,B 0,C 180,E1 -25321.989,E2 -25321.989} C_VEL
LIN {X 0,Y 143.017,Z 771.313,A -85,B 0,C 180,E1 -25324.21,E2 -25324.21} C_VEL
LIN {X 0,Y 148.11,Z 771.43,A -85,B 0,C 180,E1 -25330.938,E2 -25330.938} C_VEL
LIN {X 0,Y 151.003,Z 771.365,A -85,B 0,C 180,E1 -25332.901,E2 -25332.901} C_VEL
LIN {X 0,Y 152.232,Z 771.335,A -85,B 0,C 180,E1 -25333.479,E2 -25333.479} C_VEL
LIN {X 0,Y 162.642,Z 770.618,A -85,B 0,C 180,E1 -25337.274,E2 -25337.274} C_VEL
LIN {X 0,Y 159.307,Z 770.676,A -85,B 0,C 180,E1 -25338.567,E2 -25338.567} C_VEL
LIN {X 0,Y 149.677,Z 770.17,A -85,B 0,C 180,E1 -25342.381,E2 -25342.381} C_VEL
LIN {X 0,Y 141.186,Z 768.583,A -85,B 0,C 180,E1 -25346.8,E2 -25346.8} C_VEL
LIN {X 0,Y 133.902,Z 765.885,A -85,B 0,C 180,E1 -25351.811,E2 -25351.811} C_VEL
LIN {X 0,Y 128.375,Z 762.109,A -85,B 0,C 180,E1 -25357.466,E2 -25357.466} C_VEL
LIN {X 0,Y 124.1,Z 756.436,A -85,B 0,C 180,E1 -25364.312,E2 -25364.312} C_VEL
LIN {X 0,Y 122.181,Z 750.654,A -85,B 0,C 180,E1 -25370.063,E2 -25370.063} C_VEL
LIN {X 0,Y 121.603,Z 743.771,A -85,B 0,C 180,E1 -25375.857,E2 -25375.857} C_VEL
LIN {X 0,Y 121.499,Z 736.338,A -85,B 0,C 180,E1 -25380.828,E2 -25380.828} C_VEL
LIN {X 0,Y 121.766,Z 727.299,A -85,B 0,C 180,E1 -25385.797,E2 -25385.797} C_VEL
LIN {X 0,Y 122.173,Z 718.133,A -85,B 0,C 180,E1 -25389.937,E2 -25389.937} C_VEL
LIN {X 0,Y 122.962,Z 707.47,A -85,B 0,C 180,E1 -25393.898,E2 -25393.898} C_VEL
LIN {X 0,Y 124.194,Z 694.981,A -85,B 0,C 180,E1 -25397.708,E2 -25397.708} C_VEL
LIN {X 0,Y 125.601,Z 681.867,A -85,B 0,C 180,E1 -25400.898,E2 -25400.898} C_VEL
LIN {X 0,Y 126.775,Z 668.37,A -85,B 0,C 180,E1 -25403.481,E2 -25403.481} C_VEL
LIN {X 0,Y 128.013,Z 654.299,A -85,B 0,C 180,E1 -25405.507,E2 -25405.507} C_VEL
LIN {X 0,Y 133.047,Z 587.321,A -85,B 0,C 180,E1 -25412.782,E2 -25412.782} C_VEL
LIN {X 0,Y 130.982,Z 557.813,A -85,B 0,C 180,E1 -25416.079,E2 -25416.079} C_VEL
LIN {X 0,Y 125.49,Z 536.422,A -85,B 0,C 180,E1 -25419.007,E2 -25419.007} C_VEL
LIN {X 0,Y 123.193,Z 526.156,A -85,B 0,C 180,E1 -25425.705,E2 -25425.705} C_VEL
LIN {X 0,Y 121.947,Z 520.422,A -85,B 0,C 180,E1 -25429.71,E2 -25429.71} C_VEL
LIN {X 0,Y 121.913,Z 520.419,A -85,B 0,C 180,E1 -25434.796,E2 -25434.796} C_VEL
LIN {X 0,Y 121.94,Z 520.421,A -85,B 0,C 180,E1 -25439.828,E2 -25439.828} C_VEL
LIN {X 0,Y 121.985,Z 520.413,A -85,B 0,C 180,E1 -25446.215,E2 -25446.215} C_VEL
LIN {X 0,Y 122.051,Z 520.406,A -85,B 0,C 180,E1 -25449.788,E2 -25449.788} C_VEL
LIN {X 0,Y 122.266,Z 520.379,A -85,B 0,C 180,E1 -25456.707,E2 -25456.707} C_VEL
LIN {X 0,Y 122.458,Z 520.351,A -85,B 0,C 180,E1 -25460.086,E2 -25460.086} C_VEL
LIN {X 0,Y 122.614,Z 520.336,A -85,B 0,C 180,E1 -25466.714,E2 -25466.714} C_VEL
LIN {X 0,Y 123.046,Z 520.277,A -85,B 0,C 180,E1 -25470,E2 -25470} C_VEL
LIN {X 0,Y 122.458,Z 520.353,A -85,B 0,C 180,E1 -25476.591,E2 -25476.591} C_VEL
LIN {X 0,Y 122.458,Z 520.354,A -85,B 0,C 180,E1 -25479.914,E2 -25479.914} C_VEL
LIN {X 0,Y 122.287,Z 520.378,A -85,B 0,C 180,E1 -25483.29,E2 -25483.29} C_VEL
LIN {X 0,Y 122.053,Z 520.406,A -85,B 0,C 180,E1 -25490.212,E2 -25490.212} C_VEL
LIN {X 0,Y 121.984,Z 520.41,A -85,B 0,C 180,E1 -25493.784,E2 -25493.784} C_VEL
LIN {X 0,Y 121.942,Z 520.419,A -85,B 0,C 180,E1 -25500.174,E2 -25500.174} C_VEL
LIN {X 0,Y 121.913,Z 520.422,A -85,B 0,C 180,E1 -25506.189,E2 -25506.189} C_VEL
LIN {X 0,Y 121.898,Z 520.419,A -85,B 0,C 180,E1 -25511.452,E2 -25511.452} C_VEL
LIN {X 0,Y 122.003,Z 520.528,A -85,B 0,C 180,E1 -25514.819,E2 -25514.819} C_VEL
LIN {X 0,Y 125.399,Z 535.264,A -85,B 0,C 180,E1 -25521.044,E2 -25521.044} C_VEL
LIN {X 0,Y 128.66,Z 549.995,A -85,B 0,C 180,E1 -25526.89,E2 -25526.89} C_VEL
LIN {X 0,Y 128.431,Z 553.55,A -85,B 0,C 180,E1 -25528.166,E2 -25528.166} C_VEL
LIN {X 0,Y 129.515,Z 578.12,A -85,B 0,C 180,E1 -25530.766,E2 -25530.766} C_VEL
LIN {X 0,Y 130.331,Z 589.268,A -85,B 0,C 180,E1 -25531.956,E2 -25531.956} C_VEL
LIN {X 0,Y 126.532,Z 661.266,A -85,B 0,C 180,E1 -25540.005,E2 -25540.005} C_VEL
LIN {X 0,Y 125.633,Z 675.966,A -85,B 0,C 180,E1 -25542.102,E2 -25542.102} C_VEL
LIN {X 0,Y 124.633,Z 688.995,A -85,B 0,C 180,E1 -25544.644,E2 -25544.644} C_VEL
LIN {X 0,Y 123.772,Z 701.181,A -85,B 0,C 180,E1 -25547.706,E2 -25547.706} C_VEL
LIN {X 0,Y 123.013,Z 712.904,A -85,B 0,C 180,E1 -25551.375,E2 -25551.375} C_VEL
LIN {X 0,Y 122.499,Z 724.427,A -85,B 0,C 180,E1 -25555.888,E2 -25555.888} C_VEL
LIN {X 0,Y 122.301,Z 734.395,A -85,B 0,C 180,E1 -25560.823,E2 -25560.823} C_VEL
LIN {X 0,Y 122.266,Z 742.368,A -85,B 0,C 180,E1 -25565.773,E2 -25565.773} C_VEL
LIN {X 0,Y 122.763,Z 749.747,A -85,B 0,C 180,E1 -25571.559,E2 -25571.559} C_VEL
LIN {X 0,Y 124.28,Z 755.063,A -85,B 0,C 180,E1 -25576.424,E2 -25576.424} C_VEL
LIN {X 0,Y 127.69,Z 760.749,A -85,B 0,C 180,E1 -25582.661,E2 -25582.661} C_VEL
LIN {X 0,Y 132.81,Z 765.119,A -85,B 0,C 180,E1 -25588.442,E2 -25588.442} C_VEL
LIN {X 0,Y 139.692,Z 768.335,A -85,B 0,C 180,E1 -25593.602,E2 -25593.602} C_VEL
LIN {X 0,Y 147.964,Z 770.398,A -85,B 0,C 180,E1 -25598.132,E2 -25598.132} C_VEL
LIN {X 0,Y 157.492,Z 771.308,A -85,B 0,C 180,E1 -25602.018,E2 -25602.018} C_VEL
LIN {X 0,Y 161.155,Z 771.336,A -85,B 0,C 180,E1 -25603.262,E2 -25603.262} C_VEL
LIN {X 0,Y 161.453,Z 771.408,A -85,B 0,C 180,E1 -25604.022,E2 -25604.022} C_VEL
LIN {X 0,Y 153.778,Z 771.72,A -85,B 0,C 180,E1 -25606.722,E2 -25606.722} C_VEL
LIN {X 0,Y 144.666,Z 771.25,A -85,B 0,C 180,E1 -25610.835,E2 -25610.835} C_VEL
LIN {X 0,Y 136.931,Z 769.784,A -85,B 0,C 180,E1 -25615.627,E2 -25615.627} C_VEL
LIN {X 0,Y 130.714,Z 767.286,A -85,B 0,C 180,E1 -25621.06,E2 -25621.06} C_VEL
LIN {X 0,Y 126.197,Z 763.696,A -85,B 0,C 180,E1 -25627.056,E2 -25627.056} C_VEL
LIN {X 0,Y 123.664,Z 758.962,A -85,B 0,C 180,E1 -25633.492,E2 -25633.492} C_VEL
LIN {X 0,Y 123.013,Z 752.876,A -85,B 0,C 180,E1 -25640.131,E2 -25640.131} C_VEL
LIN {X 0,Y 123.632,Z 746.008,A -85,B 0,C 180,E1 -25645.925,E2 -25645.925} C_VEL
LIN {X 0,Y 124.073,Z 743.416,A -85,B 0,C 180,E1 -25647.971,E2 -25647.971} C_VEL
LIN {X 0,Y 122.651,Z 749.994,A -85,B 0,C 180,E1 -25653.285,E2 -25653.285} C_VEL
LIN {X 0,Y 122.243,Z 754.986,A -85,B 0,C 180,E1 -25658.264,E2 -25658.264} C_VEL
LIN {X 0,Y 122.672,Z 760.313,A -85,B 0,C 180,E1 -25664.94,E2 -25664.94} C_VEL
LIN {X 0,Y 124.083,Z 763.49,A -85,B 0,C 180,E1 -25669.867,E2 -25669.867} C_VEL
LIN {X 0,Y 127.703,Z 766.862,A -85,B 0,C 180,E1 -25676.122,E2 -25676.122} C_VEL
LIN {X 0,Y 135.059,Z 769.848,A -85,B 0,C 180,E1 -25683.635,E2 -25683.635} C_VEL
LIN {X 0,Y 143.866,Z 771.177,A -85,B 0,C 180,E1 -25689.425,E2 -25689.425} C_VEL
LIN {X 0,Y 152.232,Z 771.335,A -85,B 0,C 180,E1 -25693.479,E2 -25693.479} C_VEL
LIN {X 0,Y 153.278,Z 771.291,A -85,B 0,C 180,E1 -25694.343,E2 -25694.343} C_VEL
LIN {X 0,Y 153.187,Z 771.169,A -85,B 0,C 180,E1 -25695.652,E2 -25695.652} C_VEL
LIN {X 0,Y 151.504,Z 770.929,A -85,B 0,C 180,E1 -25697.325,E2 -25697.325} C_VEL
LIN {X 0,Y 149.384,Z 770.658,A -85,B 0,C 180,E1 -25698.56,E2 -25698.56} C_VEL
LIN {X 0,Y 143.048,Z 769.781,A -85,B 0,C 180,E1 -25701.373,E2 -25701.373} C_VEL
LIN {X 0,Y 136.812,Z 768.361,A -85,B 0,C 180,E1 -25704.334,E2 -25704.334} C_VEL
LIN {X 0,Y 131.392,Z 766.539,A -85,B 0,C 180,E1 -25707.664,E2 -25707.664} C_VEL
LIN {X 0,Y 124.67,Z 762.879,A -85,B 0,C 180,E1 -25713.193,E2 -25713.193} C_VEL
LIN {X 0,Y 119.736,Z 758.116,A -85,B 0,C 180,E1 -25719.38,E2 -25719.38} C_VEL
LIN {X 0,Y 116.469,Z 752.023,A -85,B 0,C 180,E1 -25726.033,E2 -25726.033} C_VEL
LIN {X 0,Y 115.101,Z 744.427,A -85,B 0,C 180,E1 -25732.986,E2 -25732.986} C_VEL
LIN {X 0,Y 114.855,Z 737.435,A -85,B 0,C 180,E1 -25738.247,E2 -25738.247} C_VEL
LIN {X 0,Y 114.924,Z 728.743,A -85,B 0,C 180,E1 -25743.506,E2 -25743.506} C_VEL
LIN {X 0,Y 115.309,Z 717.958,A -85,B 0,C 180,E1 -25748.764,E2 -25748.764} C_VEL
LIN {X 0,Y 115.999,Z 707.289,A -85,B 0,C 180,E1 -25753.04,E2 -25753.04} C_VEL
LIN {X 0,Y 117.098,Z 695.24,A -85,B 0,C 180,E1 -25756.968,E2 -25756.968} C_VEL
LIN {X 0,Y 118.479,Z 681.999,A -85,B 0,C 180,E1 -25760.395,E2 -25760.395} C_VEL
LIN {X 0,Y 119.673,Z 668.604,A -85,B 0,C 180,E1 -25763.125,E2 -25763.125} C_VEL
LIN {X 0,Y 120.98,Z 653.075,A -85,B 0,C 180,E1 -25765.483,E2 -25765.483} C_VEL
LIN {X 0,Y 126.006,Z 587.52,A -85,B 0,C 180,E1 -25773.132,E2 -25773.132} C_VEL
LIN {X 0,Y 123.999,Z 559.011,A -85,B 0,C 180,E1 -25776.521,E2 -25776.521} C_VEL
LIN {X 0,Y 118.225,Z 536.398,A -85,B 0,C 180,E1 -25779.703,E2 -25779.703} C_VEL
LIN {X 0,Y 115.941,Z 526.349,A -85,B 0,C 180,E1 -25786.669,E2 -25786.669} C_VEL
LIN {X 0,Y 114.867,Z 521.302,A -85,B 0,C 180,E1 -25790.454,E2 -25790.454} C_VEL
LIN {X 0,Y 114.819,Z 521.302,A -85,B 0,C 180,E1 -25796.572,E2 -25796.572} C_VEL
LIN {X 0,Y 114.872,Z 521.3,A -85,B 0,C 180,E1 -25800.695,E2 -25800.695} C_VEL
LIN {X 0,Y 114.948,Z 521.289,A -85,B 0,C 180,E1 -25806.507,E2 -25806.507} C_VEL
LIN {X 0,Y 115.02,Z 521.275,A -85,B 0,C 180,E1 -25812.211,E2 -25812.211} C_VEL
LIN {X 0,Y 115.288,Z 521.25,A -85,B 0,C 180,E1 -25817.257,E2 -25817.257} C_VEL
LIN {X 0,Y 115.394,Z 521.232,A -85,B 0,C 180,E1 -25819.472,E2 -25819.472} C_VEL
LIN {X 0,Y 115.54,Z 521.217,A -85,B 0,C 180,E1 -25826.512,E2 -25826.512} C_VEL
LIN {X 0,Y 115.999,Z 521.154,A -85,B 0,C 180,E1 -25830,E2 -25830} C_VEL
LIN {X 0,Y 115.399,Z 521.231,A -85,B 0,C 180,E1 -25836.996,E2 -25836.996} C_VEL
LIN {X 0,Y 115.394,Z 521.234,A -85,B 0,C 180,E1 -25840.528,E2 -25840.528} C_VEL
LIN {X 0,Y 115.161,Z 521.263,A -85,B 0,C 180,E1 -25844.129,E2 -25844.129} C_VEL
LIN {X 0,Y 114.983,Z 521.287,A -85,B 0,C 180,E1 -25851.514,E2 -25851.514} C_VEL
LIN {X 0,Y 114.872,Z 521.294,A -85,B 0,C 180,E1 -25855.358,E2 -25855.358} C_VEL
LIN {X 0,Y 114.869,Z 521.301,A -85,B 0,C 180,E1 -25861.068,E2 -25861.068} C_VEL
LIN {X 0,Y 114.803,Z 521.31,A -85,B 0,C 180,E1 -25867.747,E2 -25867.747} C_VEL
LIN {X 0,Y 114.94,Z 521.397,A -85,B 0,C 180,E1 -25874.239,E2 -25874.239} C_VEL
LIN {X 0,Y 118.471,Z 536.817,A -85,B 0,C 180,E1 -25881.041,E2 -25881.041} C_VEL
LIN {X 0,Y 121.477,Z 550.369,A -85,B 0,C 180,E1 -25886.659,E2 -25886.659} C_VEL
LIN {X 0,Y 121.374,Z 553.481,A -85,B 0,C 180,E1 -25887.86,E2 -25887.86} C_VEL
LIN {X 0,Y 122.344,Z 577.534,A -85,B 0,C 180,E1 -25890.612,E2 -25890.612} C_VEL
LIN {X 0,Y 123.214,Z 589.461,A -85,B 0,C 180,E1 -25891.959,E2 -25891.959} C_VEL
LIN {X 0,Y 119.69,Z 656.587,A -85,B 0,C 180,E1 -25899.967,E2 -25899.967} C_VEL
LIN {X 0,Y 118.879,Z 672.22,A -85,B 0,C 180,E1 -25902.174,E2 -25902.174} C_VEL
LIN {X 0,Y 118.017,Z 684.685,A -85,B 0,C 180,E1 -25904.552,E2 -25904.552} C_VEL
LIN {X 0,Y 117.076,Z 698.032,A -85,B 0,C 180,E1 -25907.872,E2 -25907.872} C_VEL
LIN {X 0,Y 116.417,Z 709.104,A -85,B 0,C 180,E1 -25911.32,E2 -25911.32} C_VEL
LIN {X 0,Y 115.932,Z 720.159,A -85,B 0,C 180,E1 -25915.654,E2 -25915.654} C_VEL
LIN {X 0,Y 115.718,Z 729.255,A -85,B 0,C 180,E1 -25920,E2 -25920} C_VEL
LIN {X 0,Y 115.72,Z 735.398,A -85,B 0,C 180,E1 -25923.482,E2 -25923.482} C_VEL
LIN {X 0,Y 115.787,Z 741.799,A -85,B 0,C 180,E1 -25927.849,E2 -25927.849} C_VEL
LIN {X 0,Y 116.667,Z 749.225,A -85,B 0,C 180,E1 -25933.943,E2 -25933.943} C_VEL
LIN {X 0,Y 119.273,Z 756.066,A -85,B 0,C 180,E1 -25940.704,E2 -25940.704} C_VEL
LIN {X 0,Y 123.92,Z 761.552,A -85,B 0,C 180,E1 -25946.982,E2 -25946.982} C_VEL
LIN {X 0,Y 130.092,Z 765.751,A -85,B 0,C 180,E1 -25952.7,E2 -25952.7} C_VEL
LIN {X 0,Y 138.042,Z 768.853,A -85,B 0,C 180,E1 -25957.658,E2 -25957.658} C_VEL
LIN {X 0,Y 147.274,Z 770.824,A -85,B 0,C 180,E1 -25961.92,E2 -25961.92} C_VEL
LIN {X 0,Y 150.735,Z 771.231,A -85,B 0,C 180,E1 -25963.242,E2 -25963.242} C_VEL
LIN {X 0,Y 150.248,Z 771.304,A -85,B 0,C 180,E1 -25964.281,E2 -25964.281} C_VEL
LIN {X 0,Y 139.282,Z 770.298,A -85,B 0,C 180,E1 -25969.007,E2 -25969.007} C_VEL
LIN {X 0,Y 131.24,Z 768.398,A -85,B 0,C 180,E1 -25973.91,E2 -25973.91} C_VEL
LIN {X 0,Y 124.739,Z 765.504,A -85,B 0,C 180,E1 -25979.531,E2 -25979.531} C_VEL
LIN {X 0,Y 119.999,Z 761.543,A -85,B 0,C 180,E1 -25985.797,E2 -25985.797} C_VEL
LIN {X 0,Y 117.315,Z 756.453,A -85,B 0,C 180,E1 -25992.57,E2 -25992.57} C_VEL
LIN {X 0,Y 116.649,Z 749.969,A -85,B 0,C 180,E1 -25999.587,E2 -25999.587} C_VEL
LIN {X 0,Y 117.189,Z 743.845,A -85,B 0,C 180,E1 -26004.839,E2 -26004.839} C_VEL
